// TwinCAT 3 PLC project MainPLC
// Title: IrrigationSystem
// Company: CleanGreens Solutions SA
// ProjectVersion: 0.5beat1
// ProgramVersion: 3.1.4024.0
// libraries:
//   CL_CleanGreensObjectsLibrary, * (CleanGreens SA)
//   CmpBitmapPool, * (System)
//   Tc2_Database, * (Beckhoff Automation GmbH)
//   Tc2_DataExchange, * (Beckhoff Automation GmbH)
//   Tc2_IoFunctions, * (Beckhoff Automation GmbH)
//   Tc2_Math, * (Beckhoff Automation GmbH)
//   Tc2_MC2, * (Beckhoff Automation GmbH)
//   Tc2_Standard, * (Beckhoff Automation GmbH)
//   Tc2_SUPS, * (Beckhoff Automation GmbH)
//   Tc2_System, * (Beckhoff Automation GmbH)
//   Tc2_TcpIp, * (Beckhoff Automation GmbH)
//   Tc2_Utilities, * (Beckhoff Automation GmbH)
//   Tc2_XmlDataSrv, * (Beckhoff Automation GmbH)
//   Tc3_Database, * (Beckhoff Automation GmbH)
//   Tc3_EventLogger, * (Beckhoff Automation GmbH)
//   Tc3_IotBase, * (Beckhoff Automation GmbH)
//   Tc3_IotCommunicator, * (Beckhoff Automation GmbH)
//   Tc3_JsonXml, * (Beckhoff Automation GmbH)
//   Tc3_Module, * (Beckhoff Automation GmbH)
//   VisuDialogs, * (System)
//   VisuSymbols, * (System)
//   VisuUserMgmt, * (System)
//   VisuSymbols,3.5.10.0,System
// project tree:
//   DUTs/ E_AxisErrorType.TcDUT, ST_Analog_HWI.TcDUT (not stored), ST_AXIS_MOVE_PROFILE.TcDUT, ST_CardState_HWI.TcDUT, ST_ChannelAX8206_HWI.TcDUT, ST_DriverAX8206_HWI.TcDUT, ST_PositioningLaser_HWI.TcDUT (not stored), ST_PwrSupplyAX8620_HWI.TcDUT (not stored), ST_RobotLineBoxTest_HWI.TcDUT, ST_Robot_HWI.TcDUT, ST_SystemStatus_ARP.TcDUT, ST_SystemStatus_AR.TcDUT, E_RequAxle.TcDUT, E_StepMC.TcDUT, ST_AxisMC.TcDUT, ST_Robot_Axes.TcDUT, ST_SystemStatus.TcDUT (not stored), ST_SystemStatus_ARR.TcDUT
//   GVLs/ C.TcGVL, CBot.TcGVL, G.TcGVL, GVL.TcGVL
//   / PlcTask.TcTTO
//   POUs/AxisDay2Training/ CL_Axis_old.TcPOU, FB_AxisStMachine.TcPOU, FB_AxisStMachineMaster.TcPOU
//   POUs/ CL_AxisDriverAX8206.TcPOU, CL_AxisDriverL1LeftBack.TcPOU, CL_AxisDriverL1LeftFront.TcPOU, CL_AxisDriverL2RightFront.TcPOU, CL_AxisDriverL2RightBack.TcPOU, CL_AxisMC.TcPOU, CL_AxisMCMaster.TcPOU, CL_AxisMCL2RightBack.TcPOU, CL_AxisMCL1LeftFront.TcPOU, CL_AxisMCL1LeftBack.TcPOU, CL_AxisMCL2RightFront.TcPOU, CL_CardCom.TcPOU, CL_CGSSystemBase.TcPOU, FB_testAxleAllJog.TcPOU, FB_PowerAxis1.TcPOU, FB_PowerMaster.TcPOU, FB_testAxisL1LeftFrontJog.TcPOU, FB_testAxleMasterJog.TcPOU, Main.TcPOU
// real-time tasks:
//   TASK PlcTask: cycle T#10ms, priority 20, ADS port 350
//   TASK VISU_TASK: cycle T#200000us, priority 30, ADS port 351
// motion (NC):
//   TASK NC-Task 1 SAF: cycle T#2ms, priority 4, ADS port 501
//   TASK NC-Task 1 SVB: cycle T#10ms, priority 8, ADS port 511
//   AXIS CGSMini_R01AxisL1LeftBack (id 6)
//     General: UnitName=m
//     Dynamic: AccelerationMaximum=0.5, DecelerationMaximum=1.5, Acceleration=0.3, Deceleration=1, Jerk=0.33
//     Velo: RefSearch=0.01752, RefSync=0.01752, SlowManual=0.0876, FastManual=0.5256, Fast=1.752, Maximum=0.67
//     OtherSettings: AllowMotionCmdToSlave=true
//     encoder EncType=19
//       EncPara: ScaleFactorNumerator=0.79, ScaleFactorDenominator=26214400, Inverse=true, MaxCount=#xffffffff
//         ActPosCorrection: Enable=true, Time=1
//     drive DrvType=16
//       DrvPara: Inverse=true, MaxCount=#xffffffff, DriveControlDWord=#x00020100
//         Analog: VeloReferenz=0.737, VeloScale=71.5255737304688, TorqueSetpointScale=10, ScaleFactorActTorque=0.1
//         TimeComp: TaskDelayCycles=1
//     controller CtrType=1
//       CtrPara: PriorControlFactor=1
//         PosDiffControl: Range=0.1
//         Observer: BandWidth=20
//   AXIS CGSMini_R01AxisL2RightFront (id 7)
//     General: UnitName=m
//     Dynamic: AccelerationMaximum=0.5, DecelerationMaximum=1.5, Acceleration=0.3, Deceleration=1, Jerk=0.33
//     Velo: RefSearch=0.01752, RefSync=0.01752, SlowManual=0.0876, FastManual=0.5256, Fast=1.752, Maximum=0.67
//     OtherSettings: AllowMotionCmdToSlave=true
//     encoder EncType=19
//       EncPara: ScaleFactorNumerator=0.79, ScaleFactorDenominator=26214400, Inverse=true, MaxCount=#xffffffff
//         ActPosCorrection: Enable=true, Time=1
//     drive DrvType=16
//       DrvPara: Inverse=true, MaxCount=#xffffffff, DriveControlDWord=#x00020100
//         Analog: VeloReferenz=0.737, VeloScale=71.5255737304688, TorqueSetpointScale=10, ScaleFactorActTorque=0.1
//         TimeComp: TaskDelayCycles=1
//     controller CtrType=1
//       CtrPara: PriorControlFactor=1
//         PosDiffControl: Range=0.1
//         Observer: BandWidth=20
//   AXIS CGSMini_R01AxisL2RightBack (id 8)
//     General: UnitName=m
//     Dynamic: AccelerationMaximum=0.5, DecelerationMaximum=1.5, Acceleration=0.3, Deceleration=1, Jerk=0.33
//     Velo: RefSearch=0.01752, RefSync=0.01752, SlowManual=0.0876, FastManual=0.5256, Fast=1.752, Maximum=0.67
//     OtherSettings: AllowMotionCmdToSlave=true
//     encoder EncType=19
//       EncPara: ScaleFactorNumerator=0.79, ScaleFactorDenominator=26214400, Inverse=true, MaxCount=#xffffffff
//         ActPosCorrection: Enable=true, Time=1
//     drive DrvType=16
//       DrvPara: Inverse=true, MaxCount=#xffffffff, DriveControlDWord=#x00020100
//         Analog: VeloReferenz=0.737, VeloScale=71.5255737304688, TorqueSetpointScale=10, ScaleFactorActTorque=0.1
//         TimeComp: TaskDelayCycles=1
//     controller CtrType=1
//       CtrPara: PriorControlFactor=1
//         PosDiffControl: Range=0.1
//         Observer: BandWidth=20
//   AXIS CGSMini_R01AxisL1LeftFront (id 5)
//     General: UnitName=m
//     Dynamic: AccelerationMaximum=0.5, DecelerationMaximum=1.5, Acceleration=0.3, Deceleration=1, Jerk=0.33
//     Velo: RefSearch=0.01752, RefSync=0.01752, SlowManual=0.0876, FastManual=0.5256, Fast=1.752, Maximum=0.67
//     OtherSettings: AllowMotionCmdToSlave=true
//     encoder EncType=19
//       EncPara: ScaleFactorNumerator=0.79, ScaleFactorDenominator=26214400, Inverse=true, MaxCount=#xffffffff
//         ActPosCorrection: Enable=true, Time=1
//     drive DrvType=16
//       DrvPara: Inverse=true, MaxCount=#xffffffff, DriveControlDWord=#x00020100
//         Analog: VeloReferenz=0.737, VeloScale=71.5255737304688, TorqueSetpointScale=10, ScaleFactorActTorque=0.1
//         TimeComp: TaskDelayCycles=1
//     controller CtrType=1
//       CtrPara: PriorControlFactor=1
//         PosDiffControl: Range=0.1
//         Observer: BandWidth=20
//   AXIS CGSMini_R01AxisMaster (id 14)
//     General: UnitName=m
//     Dynamic: AccelerationMaximum=0.5, DecelerationMaximum=1.5, Acceleration=0.3, Deceleration=1, Jerk=0.33
//     Velo: RefSearch=0.01752, RefSync=0.01752, SlowManual=0.0876, FastManual=0.5256, Fast=1.752, Maximum=0.67
//     OtherSettings: AllowMotionCmdToSlave=true
//     encoder EncType=1
//       EncPara: ScaleFactorNumerator=0.79, ScaleFactorDenominator=26214400, Inverse=true
//         ActPosCorrection: Enable=true, Time=1
//     drive DrvType=5
//       DrvPara: Inverse=true
//         Analog: VeloReferenz=0.737, TorqueSetpointScale=10, ScaleFactorActTorque=0.1
//         TimeComp: TaskDelayCycles=1
//     controller CtrType=1
//       CtrPara: PriorControlFactor=1
//         PosDiffControl: Range=0.1
//         Observer: BandWidth=20
//   AXIS Sim_Robot01AxisLine1Back (id 9)
//     OtherSettings: AllowMotionCmdToSlave=true
//     encoder EncType=1
//     drive DrvType=5
//       Analog: TorqueSetpointScale=10, ScaleFactorActTorque=0.1
//       TimeComp: TaskDelayCycles=1
//     controller CtrType=1
//       CtrPara: PriorControlFactor=1
//         Observer: BandWidth=20
//   AXIS Sim_Robot01AxisLine2Back (id 10)
//     OtherSettings: AllowMotionCmdToSlave=true
//     encoder EncType=1
//     drive DrvType=5
//       Analog: TorqueSetpointScale=10, ScaleFactorActTorque=0.1
//       TimeComp: TaskDelayCycles=1
//     controller CtrType=1
//       CtrPara: PriorControlFactor=1
//         Observer: BandWidth=20
//   AXIS Sim_Robot01AxisLine1Front (id 11)
//     OtherSettings: AllowMotionCmdToSlave=true
//     encoder EncType=1
//     drive DrvType=5
//       Analog: TorqueSetpointScale=10, ScaleFactorActTorque=0.1
//       TimeComp: TaskDelayCycles=1
//     controller CtrType=1
//       CtrPara: PriorControlFactor=1
//         Observer: BandWidth=20
//   AXIS Sim_Robot01AxisLine2Front (id 12)
//     OtherSettings: AllowMotionCmdToSlave=true
//     encoder EncType=1
//     drive DrvType=5
//       Analog: TorqueSetpointScale=10, ScaleFactorActTorque=0.1
//       TimeComp: TaskDelayCycles=1
//     controller CtrType=1
//       CtrPara: PriorControlFactor=1
//         Observer: BandWidth=20
//   AXIS Sim_Robot01AxisMaster (id 13)
//     OtherSettings: AllowMotionCmdToSlave=true
//     encoder EncType=1
//     drive DrvType=5
//       Analog: TorqueSetpointScale=10, ScaleFactorActTorque=0.1
//       TimeComp: TaskDelayCycles=1
//     controller CtrType=1
//       CtrPara: PriorControlFactor=1
//         Observer: BandWidth=20
// I/O:
//   DEVICE CGSMini_IRSMainPLCSafe, AmsNetId 5.93.147.0.2.1
//     CGSMini_RobotAllMainCab-EL1200 [EK1200-5000 EtherCAT Power supply (2A E-Bus)]
//       CGSMini_RobotAllLicenses-EL6070 [EL6070 1Ch. Licensing-Terminal]
//       CGSMini_Robot01LineBoxOverCurrProt1-EL9222 [EL9222-5500 Overcurrent protection 24V DC, 2Ch., max. 10A (sum), adjustable]
//       CGSMini_Robot01LineBoxOutN01-EL2008 [EL2008 8Ch. Dig. Output 24V, 0.5A]
//       CGSMini_RobotAllMainCabInN01-EL1008 [EL1008 8Ch. Dig. Input 24V, 3ms]
//       CGSMini_Robot01LineBoxInN01-EL1008 [EL1008 8Ch. Dig. Input 24V, 3ms]
//       CGSMini_Robot01LineBoxAnaInN01-EL3202 [EL3202 2Ch. Ana. Input PT100 (RTD)]
//       CGSMini_Robot01LineBoxAnaInN02-EL3054 [EL3054 4Ch. Ana. Input 4-20mA]
//       CGSMini_Robot01LineBoxAnaInN03-EL3202 [EL3202 2Ch. Ana. Input PT100 (RTD)]
//       CGSMini_Robot01LineBoxSafeInN01-EL1918 [EL1918, 8Ch. Safety Input 24V, TwinSAFE] (disabled)
//         modules: Module 1 (FSOE), Module 2 (FSLOGIC)
//       CGSMini_Robot01LineBoxInN02-EL1004tmp [EL1004 4Ch. Dig. Input 24V, 3ms]
//       CGSMini_Robot01LineBoxInN03-EL1004tmp [EL1004 4Ch. Dig. Input 24V, 3ms]
//       CGSMini_RobotAllMainCabAnaInN01-EL3443 [EL3443 3Ch. Power Measuring]
//       CGSMini_Robot01MainCabEtherCATBusEK1122 [EK1122 2 port EtherCAT junction]
//         CGSMini_Robot01Laser-SickDL100 [DL100]
//         CGSMini_Robot01OnboardBox-EK1100 [EK1100 EtherCAT Coupler (2A E-Bus)]
//           CGSMini_Robot01OnBoardBoxOutN01-EL2008 [EL2008 8Ch. Dig. Output 24V, 0.5A]
//           CGSMini_Robot01OnBoardBoxAnaInN04-EL3054 [EL3054 4Ch. Ana. Input 4-20mA]
//           CGSMini_Robot01OnBoardBoxEndBus-EL9011 [EL9011 End Terminal]
//         CGSMini_Robot01OnboardAxisPwrSupply-AX8620 [AX8620-0000-0105]
//           CGSMini_Robot01OnboardAxisDriverL2Right-AX8206 [AX8206-0200-0104 (2Ch. 6A servo axis, safe-motion)]
//             modules: Device, Device, Device, Device, Device, Device, Device, Device, Device, Device, Device (Safety), Device, Device, Device, Device, Device, Device, Device, Device, Device, Device, Device, Device, Device, Device, Device, Device, Device, Device, Device, Device, Back, Back, Back, Back, Back, Back, Back, Back, Back, Back, Back, Back, Back, Back, Back, Back, Back, Back, Back, Back, Back, Back, Back, Back, Back, Back, Back, Front, Front, Front, Front, Front, Front, Front, Front, Front, Front, Front, Front, Front, Front, Front, Front, Front, Front, Front, Front, Front, Front, Front, Front, Front, Front, Front
//             startup 12992:1 := 414D383733312D78437830 // Ch A Motor parameters / Configured motor type
//             startup 24768:0 := FEFF // Ch A Interpolation sub mode select
//             startup 13000:5 := 0200 // Ch A Motor thermal model / Reaction
//             startup 13000:6 := 0000C841 // Ch A Motor thermal model / Partial fraction factor
//             startup 12992:12 := 00803B45 // Ch A Motor parameters / Motor rated speed
//             startup 12992:13 := 8D97A63F // Ch A Motor parameters / Motor rated torque
//             startup 24694:0 := 5A050000 // Ch A Motor standstill torque
//             startup 24800:0 := D007 // Ch A Positive torque/force limit value
//             startup 24801:0 := D007 // Ch A Negative torque/force limit value
//             startup 12288:6 := 4158383230362D303230302D30303030 // Ch A AxisMain parameters / Configured drive type
//             startup 12867:1 := 0000803F // Ch A TorqueCtrl parameters / Configured channel rated current
//             startup 12867:2 := 00004040 // Ch A TorqueCtrl parameters / Configured channel peak current
//             startup 24672:0 := 08 // Ch A Modes of operation
//             startup 12864:1 := 0D4DF043 // Ch A TorqueCtrl parameters mappable / Torque control proportional gain q
//             startup 12864:2 := 8A0E7C39 // Ch A TorqueCtrl parameters mappable / Torque control integral action time q
//             startup 12608:1 := 3C03B63C // Ch A VeloCtrl parameters mappable / Velocity control proportional gain
//             startup 12608:2 := 6F12033C // Ch A VeloCtrl parameters mappable / Velocity control integral action time
//             startup 12608:3 := 00701446 // Ch A VeloCtrl parameters mappable / Bipolar velocity limit value
//             startup 12992:15 := 0100 // Ch A Motor parameters / Motor temperature sensor connection
//             startup 12611:4 := 0400 // Ch A VeloCtrl observer / Observer type
//             startup 24672:0 := 08 // Ch A Modes of operation
//             startup 12296:2 := 00 // Ch A AxisMain parameters encoder polarity / Primary encoder actual values
//             startup 14016:1 := 414D383733312D78437830 // Ch B Motor parameters / Configured motor type
//             startup 26816:0 := FEFF // Ch B Interpolation sub mode select
//             startup 14024:5 := 0200 // Ch B Motor thermal model / Reaction
//             startup 14024:6 := 0000C841 // Ch B Motor thermal model / Partial fraction factor
//             startup 14016:12 := 00803B45 // Ch B Motor parameters / Motor rated speed
//             startup 14016:13 := 8D97A63F // Ch B Motor parameters / Motor rated torque
//             startup 26742:0 := 5A050000 // Ch B Motor standstill torque
//             startup 26848:0 := D007 // Ch B Positive torque/force limit value
//             startup 26849:0 := D007 // Ch B Negative torque/force limit value
//             startup 13312:6 := 4158383230362D303230302D30303030 // Ch B AxisMain parameters / Configured drive type
//             startup 13891:1 := 0000803F // Ch B TorqueCtrl parameters / Configured channel rated current
//             startup 13891:2 := 00004040 // Ch B TorqueCtrl parameters / Configured channel peak current
//             startup 26720:0 := 08 // Ch B Modes of operation
//             startup 13888:1 := 0D4DF043 // Ch B TorqueCtrl parameters mappable / Torque control proportional gain q
//             startup 13888:2 := 8A0E7C39 // Ch B TorqueCtrl parameters mappable / Torque control integral action time q
//             startup 13632:1 := 3C03B63C // Ch B VeloCtrl parameters mappable / Velocity control proportional gain
//             startup 13632:2 := 6F12033C // Ch B VeloCtrl parameters mappable / Velocity control integral action time
//             startup 13632:3 := 00701446 // Ch B VeloCtrl parameters mappable / Bipolar velocity limit value
//             startup 14016:15 := 0100 // Ch B Motor parameters / Motor temperature sensor connection
//             startup 13635:4 := 0400 // Ch B VeloCtrl observer / Observer type
//             startup 26720:0 := 08 // Ch B Modes of operation
//             startup 13320:2 := 00 // Ch B AxisMain parameters encoder polarity / Primary encoder actual values
//           CGSMini_Robot01OnboardAxisDriverL1Left-AX8206 [AX8206-0200-0104 (2Ch. 6A servo axis, safe-motion)]
//             modules: Device, Device, Device, Device, Device, Device, Device, Device, Device, Device, Device (Safety), Device, Device, Device, Device, Device, Device, Device, Device, Device, Device, Device, Device, Device, Device, Device, Device, Device, Device, Device, Device, Back, Back, Back, Back, Back, Back, Back, Back, Back, Back, Back, Back, Back, Back, Back, Back, Back, Back, Back, Back, Back, Back, Back, Back, Back, Back, Back, Front, Front, Front, Front, Front, Front, Front, Front, Front, Front, Front, Front, Front, Front, Front, Front, Front, Front, Front, Front, Front, Front, Front, Front, Front, Front, Front
//             startup 12992:1 := 414D383733312D78437830 // Ch A Motor parameters / Configured motor type
//             startup 24768:0 := FEFF // Ch A Interpolation sub mode select
//             startup 13000:5 := 0200 // Ch A Motor thermal model / Reaction
//             startup 13000:6 := 0000C841 // Ch A Motor thermal model / Partial fraction factor
//             startup 12992:12 := 00803B45 // Ch A Motor parameters / Motor rated speed
//             startup 12992:13 := 8D97A63F // Ch A Motor parameters / Motor rated torque
//             startup 24694:0 := 5A050000 // Ch A Motor standstill torque
//             startup 24800:0 := D007 // Ch A Positive torque/force limit value
//             startup 24801:0 := D007 // Ch A Negative torque/force limit value
//             startup 12288:6 := 4158383230362D303230302D30303030 // Ch A AxisMain parameters / Configured drive type
//             startup 12867:1 := 0000803F // Ch A TorqueCtrl parameters / Configured channel rated current
//             startup 12867:2 := 00004040 // Ch A TorqueCtrl parameters / Configured channel peak current
//             startup 24672:0 := 08 // Ch A Modes of operation
//             startup 12864:1 := 0D4DF043 // Ch A TorqueCtrl parameters mappable / Torque control proportional gain q
//             startup 12864:2 := 8A0E7C39 // Ch A TorqueCtrl parameters mappable / Torque control integral action time q
//             startup 12608:1 := 3C03B63C // Ch A VeloCtrl parameters mappable / Velocity control proportional gain
//             startup 12608:2 := 6F12033C // Ch A VeloCtrl parameters mappable / Velocity control integral action time
//             startup 12608:3 := 00701446 // Ch A VeloCtrl parameters mappable / Bipolar velocity limit value
//             startup 12992:15 := 0100 // Ch A Motor parameters / Motor temperature sensor connection
//             startup 12611:4 := 0400 // Ch A VeloCtrl observer / Observer type
//             startup 24672:0 := 08 // Ch A Modes of operation
//             startup 12296:2 := 00 // Ch A AxisMain parameters encoder polarity / Primary encoder actual values
//             startup 14016:1 := 414D383733312D78437830 // Ch B Motor parameters / Configured motor type
//             startup 26816:0 := FEFF // Ch B Interpolation sub mode select
//             startup 14024:5 := 0200 // Ch B Motor thermal model / Reaction
//             startup 14024:6 := 0000C841 // Ch B Motor thermal model / Partial fraction factor
//             startup 14016:12 := 00803B45 // Ch B Motor parameters / Motor rated speed
//             startup 14016:13 := 8D97A63F // Ch B Motor parameters / Motor rated torque
//             startup 26742:0 := 5A050000 // Ch B Motor standstill torque
//             startup 26848:0 := D007 // Ch B Positive torque/force limit value
//             startup 26849:0 := D007 // Ch B Negative torque/force limit value
//             startup 13312:6 := 4158383230362D303230302D30303030 // Ch B AxisMain parameters / Configured drive type
//             startup 13891:1 := 0000803F // Ch B TorqueCtrl parameters / Configured channel rated current
//             startup 13891:2 := 00004040 // Ch B TorqueCtrl parameters / Configured channel peak current
//             startup 26720:0 := 08 // Ch B Modes of operation
//             startup 13888:1 := 0D4DF043 // Ch B TorqueCtrl parameters mappable / Torque control proportional gain q
//             startup 13888:2 := 8A0E7C39 // Ch B TorqueCtrl parameters mappable / Torque control integral action time q
//             startup 13632:1 := 3C03B63C // Ch B VeloCtrl parameters mappable / Velocity control proportional gain
//             startup 13632:2 := 6F12033C // Ch B VeloCtrl parameters mappable / Velocity control integral action time
//             startup 13632:3 := 00701446 // Ch B VeloCtrl parameters mappable / Bipolar velocity limit value
//             startup 14016:15 := 0100 // Ch B Motor parameters / Motor temperature sensor connection
//             startup 13635:4 := 0400 // Ch B VeloCtrl observer / Observer type
//             startup 26720:0 := 08 // Ch B Modes of operation
//             startup 13320:2 := 00 // Ch B AxisMain parameters encoder polarity / Primary encoder actual values
//           CGSMini_Robot01OnBoardBoxEndBus1-EL9011 [EL9011 End Terminal]
// variable links:
//   MainPLC/MainPLC Instance <-> CGSMini_IRSMainPLCSafe/CGSMini_RobotAllMainCab-EL1200/CGSMini_Robot01LineBoxAnaInN01-EL3202
//     PlcTask Inputs/G.stBoxIN/stAnaInN01_3202State/bNotValid <-> WcState/WcState
//     PlcTask Inputs/G.stBoxIN/stAnaInN01_3202State/uiDataState <-> InfoData/State
//   MainPLC/MainPLC Instance <-> CGSMini_IRSMainPLCSafe/CGSMini_RobotAllMainCab-EL1200/CGSMini_Robot01LineBoxAnaInN02-EL3054
//     PlcTask Inputs/G.stBoxIN/stAnaInN02_3054State/bNotValid <-> WcState/WcState
//     PlcTask Inputs/G.stBoxIN/stAnaInN02_3054State/uiDataState <-> InfoData/State
//   MainPLC/MainPLC Instance <-> CGSMini_IRSMainPLCSafe/CGSMini_RobotAllMainCab-EL1200/CGSMini_Robot01LineBoxAnaInN03-EL3202
//     PlcTask Inputs/G.stBoxIN/stAnaInN03_3202State/bNotValid <-> WcState/WcState
//     PlcTask Inputs/G.stBoxIN/stAnaInN03_3202State/uiDataState <-> InfoData/State
//   MainPLC/MainPLC Instance <-> CGSMini_IRSMainPLCSafe/CGSMini_RobotAllMainCab-EL1200/CGSMini_Robot01LineBoxInN01-EL1008
//     PlcTask Inputs/G.stBoxIN/stInN01_1008State/bNotValid <-> WcState/WcState
//     PlcTask Inputs/G.stBoxIN/stInN01_1008State/uiDataState <-> InfoData/State
//   MainPLC/MainPLC Instance <-> CGSMini_IRSMainPLCSafe/CGSMini_RobotAllMainCab-EL1200/CGSMini_Robot01LineBoxInN02-EL1004tmp
//     PlcTask Inputs/G.stBoxIN/stInN02_1004State/bNotValid <-> WcState/WcState
//     PlcTask Inputs/G.stBoxIN/stInN02_1004State/uiDataState <-> InfoData/State
//   MainPLC/MainPLC Instance <-> CGSMini_IRSMainPLCSafe/CGSMini_RobotAllMainCab-EL1200/CGSMini_Robot01LineBoxInN03-EL1004tmp
//     PlcTask Inputs/G.stBoxIN/stInN03_1004State/bNotValid <-> WcState/WcState
//     PlcTask Inputs/G.stBoxIN/stInN03_1004State/uiDataState <-> InfoData/State
//   MainPLC/MainPLC Instance <-> CGSMini_IRSMainPLCSafe/CGSMini_RobotAllMainCab-EL1200/CGSMini_Robot01LineBoxOutN01-EL2008
//     PlcTask Inputs/G.stBoxIN/stOutN01_2008State/bNotValid <-> WcState/WcState
//     PlcTask Inputs/G.stBoxIN/stOutN01_2008State/uiDataState <-> InfoData/State
//   MainPLC/MainPLC Instance <-> CGSMini_IRSMainPLCSafe/CGSMini_RobotAllMainCab-EL1200/CGSMini_Robot01LineBoxOverCurrProt1-EL9222
//     PlcTask Inputs/G.stBoxIN/stOverCProt1_9222State/bNotValid <-> WcState/WcState
//     PlcTask Inputs/G.stBoxIN/stOverCProt1_9222State/uiDataState <-> InfoData/State
//   MainPLC/MainPLC Instance <-> CGSMini_IRSMainPLCSafe/CGSMini_RobotAllMainCab-EL1200/CGSMini_Robot01LineBoxSafeInN01-EL1918
//     PlcTask Inputs/G.stBoxIN/stSafety_1918State/bNotValid <-> WcState/WcState
//     PlcTask Inputs/G.stBoxIN/stSafety_1918State/uiDataState <-> InfoData/State
//   MainPLC/MainPLC Instance <-> CGSMini_IRSMainPLCSafe/CGSMini_RobotAllMainCab-EL1200/CGSMini_Robot01MainCabEtherCATBusEK1122/CGSMini_Robot01Laser-SickDL100
//     PlcTask Inputs/G.stBoxIN/stLaserPos_State/bNotValid <-> WcState/WcState
//     PlcTask Inputs/G.stBoxIN/stLaserPos_State/uiDataState <-> InfoData/State
//     PlcTask Inputs/G.stIN/stLaserPos <-> Distance/Distance
//     PlcTask Inputs/G.stIN/stLaserPos_State/bNotValid <-> WcState/WcState
//     PlcTask Inputs/G.stIN/stLaserPos_State/uiDataState <-> InfoData/State
//   MainPLC/MainPLC Instance <-> CGSMini_IRSMainPLCSafe/CGSMini_RobotAllMainCab-EL1200/CGSMini_Robot01MainCabEtherCATBusEK1122/CGSMini_Robot01OnboardAxisPwrSupply-AX8620
//     PlcTask Inputs/G.stIN/stPwrSupplyAX8620/comState/bNotValid <-> WcState/WcState
//     PlcTask Inputs/G.stIN/stPwrSupplyAX8620/comState/uiDataState <-> InfoData/State
//     PlcTask Inputs/G.stIN/stPwrSupplyAX8620/sdiDcInputShift <-> InfoData/DcInputShift
//     PlcTask Inputs/G.stIN/stPwrSupplyAX8620/sdiDcOutputShift <-> InfoData/DcOutputShift
//   MainPLC/MainPLC Instance <-> CGSMini_IRSMainPLCSafe/CGSMini_RobotAllMainCab-EL1200/CGSMini_Robot01MainCabEtherCATBusEK1122/CGSMini_Robot01OnboardAxisPwrSupply-AX8620/CGSMini_Robot01OnboardAxisDriverL1Left-AX8206
//     PlcTask Inputs/G.stIN/stDriverL1Left/comState <-> InfoData/State
//     PlcTask Inputs/G.stIN/stDriverL1Left/sdiDcInputShift <-> InfoData/DcInputShift
//     PlcTask Inputs/G.stIN/stDriverL1Left/sdiDcOutputShift <-> InfoData/DcOutputShift
//   MainPLC/MainPLC Instance <-> CGSMini_IRSMainPLCSafe/CGSMini_RobotAllMainCab-EL1200/CGSMini_Robot01MainCabEtherCATBusEK1122/CGSMini_Robot01OnboardAxisPwrSupply-AX8620/CGSMini_Robot01OnboardAxisDriverL2Right-AX8206
//     PlcTask Inputs/G.stIN/stDriverL2Right/comState <-> InfoData/State
//     PlcTask Inputs/G.stIN/stDriverL2Right/sdiDcInputShift <-> InfoData/DcInputShift
//     PlcTask Inputs/G.stIN/stDriverL2Right/sdiDcOutputShift <-> InfoData/DcOutputShift
//   MainPLC/MainPLC Instance <-> CGSMini_IRSMainPLCSafe/CGSMini_RobotAllMainCab-EL1200/CGSMini_Robot01MainCabEtherCATBusEK1122/CGSMini_Robot01OnboardBox-EK1100
//     PlcTask Inputs/G.stIN/stOnboardBox_1100State/uiDataState <-> InfoData/State
//   MainPLC/MainPLC Instance <-> CGSMini_IRSMainPLCSafe/CGSMini_RobotAllMainCab-EL1200/CGSMini_Robot01MainCabEtherCATBusEK1122/CGSMini_Robot01OnboardBox-EK1100/CGSMini_Robot01OnBoardBoxAnaInN04-EL3054
//     PlcTask Inputs/G.stIN/stAnaInN04_3054State/bNotValid <-> WcState/WcState
//     PlcTask Inputs/G.stIN/stAnaInN04_3054State/uiDataState <-> InfoData/State
//     PlcTask Inputs/G.stIN/stAnaOnboardSpare1/bTError <-> Spare1/Status/Error
//     PlcTask Inputs/G.stIN/stAnaOnboardSpare1/bTLimit1 <-> Spare1/Status/Limit 1
//     PlcTask Inputs/G.stIN/stAnaOnboardSpare1/bTLimit2 <-> Spare1/Status/Limit 2
//     PlcTask Inputs/G.stIN/stAnaOnboardSpare1/bTOverRange <-> Spare1/Status/Overrange
//     PlcTask Inputs/G.stIN/stAnaOnboardSpare1/bTUnderRange <-> Spare1/Status/Underrange
//     PlcTask Inputs/G.stIN/stAnaOnboardSpare1/siAnaRaw <-> Spare1/Value
//   MainPLC/MainPLC Instance <-> CGSMini_IRSMainPLCSafe/CGSMini_RobotAllMainCab-EL1200/CGSMini_Robot01MainCabEtherCATBusEK1122/CGSMini_Robot01OnboardBox-EK1100/CGSMini_Robot01OnBoardBoxOutN01-EL2008
//     PlcTask Inputs/G.stIN/stOutN01_2008State/bNotValid <-> WcState/WcState
//     PlcTask Inputs/G.stIN/stOutN01_2008State/uiDataState <-> InfoData/State
//   MainPLC/MainPLC Instance <-> NC-Task 1 SAF/Axes/CGSMini_R01AxisL1LeftBack
//     PlcTask Inputs/G.stAX.L1LeftBack.NcToPlc <-> Outputs/ToPlc
//     PlcTask Outputs/G.stAX.L1LeftBack.PlcToNc <-> Inputs/FromPlc
//   MainPLC/MainPLC Instance <-> NC-Task 1 SAF/Axes/CGSMini_R01AxisL1LeftFront
//     PlcTask Inputs/G.stAX.L1LeftFront.NcToPlc <-> Outputs/ToPlc
//     PlcTask Outputs/G.stAX.L1LeftFront.PlcToNc <-> Inputs/FromPlc
//   MainPLC/MainPLC Instance <-> NC-Task 1 SAF/Axes/CGSMini_R01AxisL2RightBack
//     PlcTask Inputs/G.stAX.L2RightBack.NcToPlc <-> Outputs/ToPlc
//     PlcTask Outputs/G.stAX.L2RightBack.PlcToNc <-> Inputs/FromPlc
//   MainPLC/MainPLC Instance <-> NC-Task 1 SAF/Axes/CGSMini_R01AxisL2RightFront
//     PlcTask Inputs/G.stAX.L2RightFront.NcToPlc <-> Outputs/ToPlc
//     PlcTask Outputs/G.stAX.L2RightFront.PlcToNc <-> Inputs/FromPlc
//   MainPLC/MainPLC Instance <-> NC-Task 1 SAF/Axes/CGSMini_R01AxisMaster
//     PlcTask Inputs/G.stAX.Master.NcToPlc <-> Outputs/ToPlc
//     PlcTask Outputs/G.stAX.Master.PlcToNc <-> Inputs/FromPlc
//   (this object) <-> CGSMini_IRSMainPLCSafe/CGSMini_RobotAllMainCab-EL1200/CGSMini_Robot01MainCabEtherCATBusEK1122/CGSMini_Robot01OnboardAxisPwrSupply-AX8620/CGSMini_Robot01OnboardAxisDriverL1Left-AX8206
//     Drive/Inputs/In/nDataIn1 <-> Back/Ch A PositionControl Inputs/Ch A Following error actual value
//     Drive/Inputs/In/nDcOutputTime <-> InfoData/DcOutputShift
//     Drive/Inputs/In/nState1 <-> Back/Ch A AxisMain Inputs/Ch A Statusword
//     Drive/Inputs/In/nState2 <-> Back/Ch A AxisMain Inputs/Ch A Statusword @bit 8
//     Drive/Outputs/Out/nCtrl1 <-> Back/Ch A AxisMain Outputs/Ch A Controlword
//     Drive/Outputs/Out/nCtrl2 <-> Back/Ch A AxisMain Outputs/Ch A Controlword @bit 8
//     Drive/Outputs/Out/nDataOut1 <-> Back/Ch A Interpolator Outputs/Ch A Target position
//     Drive/Outputs/Out/nDataOut2 <-> Back/Ch A Interpolator Outputs/Ch A Target velocity
//     Enc/Inputs/In/nDataIn1 <-> Back/Ch A AxisMain Inputs/Ch A Position actual value
//     Enc/Inputs/In/nDcInputTime <-> InfoData/DcInputShift
//     Enc/Inputs/In/nState2 @bit 5 <-> Back/Ch A AxisMain Inputs/Position actual value invalid
//     Drive/Inputs/In/nDataIn1 <-> Front/Ch B PositionControl Inputs/Ch B Following error actual value
//     Drive/Inputs/In/nState1 <-> Front/Ch B AxisMain Inputs/Ch B Statusword
//     Drive/Inputs/In/nState2 <-> Front/Ch B AxisMain Inputs/Ch B Statusword @bit 8
//     Drive/Outputs/Out/nCtrl1 <-> Front/Ch B AxisMain Outputs/Ch B Controlword
//     Drive/Outputs/Out/nCtrl2 <-> Front/Ch B AxisMain Outputs/Ch B Controlword @bit 8
//     Drive/Outputs/Out/nDataOut1 <-> Front/Ch B Interpolator Outputs/Ch B Target position
//     Drive/Outputs/Out/nDataOut2 <-> Front/Ch B Interpolator Outputs/Ch B Target velocity
//     Enc/Inputs/In/nDataIn1 <-> Front/Ch B AxisMain Inputs/Ch B Position actual value
//     Enc/Inputs/In/nState2 @bit 5 <-> Front/Ch B AxisMain Inputs/Position actual value invalid
//   (this object) <-> CGSMini_IRSMainPLCSafe/CGSMini_RobotAllMainCab-EL1200/CGSMini_Robot01MainCabEtherCATBusEK1122/CGSMini_Robot01OnboardAxisPwrSupply-AX8620/CGSMini_Robot01OnboardAxisDriverL2Right-AX8206
//     Drive/Inputs/In/nDataIn1 <-> Front/Ch B PositionControl Inputs/Ch B Following error actual value
//     Drive/Inputs/In/nDcOutputTime <-> InfoData/DcOutputShift
//     Drive/Inputs/In/nState1 <-> Front/Ch B AxisMain Inputs/Ch B Statusword
//     Drive/Inputs/In/nState2 <-> Front/Ch B AxisMain Inputs/Ch B Statusword @bit 8
//     Drive/Outputs/Out/nCtrl1 <-> Front/Ch B AxisMain Outputs/Ch B Controlword
//     Drive/Outputs/Out/nCtrl2 <-> Front/Ch B AxisMain Outputs/Ch B Controlword @bit 8
//     Drive/Outputs/Out/nDataOut1 <-> Front/Ch B Interpolator Outputs/Ch B Target position
//     Drive/Outputs/Out/nDataOut2 <-> Front/Ch B Interpolator Outputs/Ch B Target velocity
//     Enc/Inputs/In/nDataIn1 <-> Front/Ch B AxisMain Inputs/Ch B Position actual value
//     Enc/Inputs/In/nDcInputTime <-> InfoData/DcInputShift
//     Enc/Inputs/In/nState2 @bit 5 <-> Front/Ch B AxisMain Inputs/Position actual value invalid
//     Drive/Inputs/In/nDataIn1 <-> Back/Ch A PositionControl Inputs/Ch A Following error actual value
//     Drive/Inputs/In/nState1 <-> Back/Ch A AxisMain Inputs/Ch A Statusword
//     Drive/Inputs/In/nState2 <-> Back/Ch A AxisMain Inputs/Ch A Statusword @bit 8
//     Drive/Outputs/Out/nCtrl1 <-> Back/Ch A AxisMain Outputs/Ch A Controlword
//     Drive/Outputs/Out/nCtrl2 <-> Back/Ch A AxisMain Outputs/Ch A Controlword @bit 8
//     Drive/Outputs/Out/nDataOut1 <-> Back/Ch A Interpolator Outputs/Ch A Target position
//     Drive/Outputs/Out/nDataOut2 <-> Back/Ch A Interpolator Outputs/Ch A Target velocity
//     Enc/Inputs/In/nDataIn1 <-> Back/Ch A AxisMain Inputs/Ch A Position actual value
//     Enc/Inputs/In/nState2 @bit 5 <-> Back/Ch A AxisMain Inputs/Position actual value invalid
//   __THIS__ <-> MainPLC/MainPLC Instance
//     Inputs/FromPlc <-> PlcTask Outputs/G.stAxes.Line1Back.PlcToNc
//     Inputs/FromPlc <-> PlcTask Outputs/G.stAxes.Line2Back.PlcToNc
//     Outputs/ToPlc <-> PlcTask Inputs/G.stAxes.Line1Back.NcToPlc
//     Outputs/ToPlc <-> PlcTask Inputs/G.stAxes.Line2Back.NcToPlc
//     Inputs/FromPlc <-> PlcTask Outputs/GIQ_Robot01.stAxes.Line1Back.PlcToNc
//     Inputs/FromPlc <-> PlcTask Outputs/GIQ_Robot01.stAxes.Line2Back.PlcToNc
//     Outputs/ToPlc <-> PlcTask Inputs/GIQ_Robot01.stAxes.Line1Back.NcToPlc
//     Outputs/ToPlc <-> PlcTask Inputs/GIQ_Robot01.stAxes.Line2Back.NcToPlc
//     Inputs/FromPlc <-> PlcTask Outputs/G.stAxes.Line1Front.PlcToNc
//     Inputs/FromPlc <-> PlcTask Outputs/G.stAxes.Line2Front.PlcToNc
//     Outputs/ToPlc <-> PlcTask Inputs/G.stAxes.Line1Front.NcToPlc
//     Outputs/ToPlc <-> PlcTask Inputs/G.stAxes.Line2Front.NcToPlc
//     Inputs/FromPlc <-> PlcTask Outputs/GIQ_Robot01.stAxes.Line1Front.PlcToNc
//     Inputs/FromPlc <-> PlcTask Outputs/GIQ_Robot01.stAxes.Line2Front.PlcToNc
//     Outputs/ToPlc <-> PlcTask Inputs/GIQ_Robot01.stAxes.Line1Front.NcToPlc
//     Outputs/ToPlc <-> PlcTask Inputs/GIQ_Robot01.stAxes.Line2Front.NcToPlc
//     Inputs/FromPlc <-> PlcTask Outputs/G.stAxes.Master.PlcToNc
//     Outputs/ToPlc <-> PlcTask Inputs/G.stAxes.Master.NcToPlc
//   (this object) <-> MainPLC/MainPLC Instance
//     Inputs/FromPlc <-> PlcTask Outputs/G.stAxes.Line1Back.PlcToNc
//     Inputs/FromPlc <-> PlcTask Outputs/G.stAxes.Line2Back.PlcToNc
//     Outputs/ToPlc <-> PlcTask Inputs/G.stAxes.Line1Back.NcToPlc
//     Outputs/ToPlc <-> PlcTask Inputs/G.stAxes.Line2Back.NcToPlc
//     Inputs/FromPlc <-> PlcTask Outputs/G.stAxes.Line1Front.PlcToNc
//     Inputs/FromPlc <-> PlcTask Outputs/G.stAxes.Line2Front.PlcToNc
//     Outputs/ToPlc <-> PlcTask Inputs/G.stAxes.Line1Front.NcToPlc
//     Outputs/ToPlc <-> PlcTask Inputs/G.stAxes.Line2Front.NcToPlc
//     Inputs/FromPlc <-> PlcTask Outputs/G.stAxes.Master.PlcToNc
//     Outputs/ToPlc <-> PlcTask Inputs/G.stAxes.Master.NcToPlc
//   (this object) <-> CGSMini_IRSMainPLCSafe
//     CGSMini_RobotAllMainCab-EL1200/CGSMini_Robot01MainCabEtherCATBusEK1122/CGSMini_Robot01OnboardAxisPwrSupply-AX8620/CGSMini_Robot01OnboardAxisDriverL1Left-AX8206/Device/DeviceMain Outputs/Power supply controlword <-> CGSMini_RobotAllMainCab-EL1200/CGSMini_Robot01MainCabEtherCATBusEK1122/CGSMini_Robot01OnboardAxisPwrSupply-AX8620/PSM Controlword for axis/Controlword for axis
//     CGSMini_RobotAllMainCab-EL1200/CGSMini_Robot01MainCabEtherCATBusEK1122/CGSMini_Robot01OnboardAxisPwrSupply-AX8620/CGSMini_Robot01OnboardAxisDriverL2Right-AX8206/Device/DeviceMain Outputs/Power supply controlword <-> CGSMini_RobotAllMainCab-EL1200/CGSMini_Robot01MainCabEtherCATBusEK1122/CGSMini_Robot01OnboardAxisPwrSupply-AX8620/PSM Controlword for axis/Controlword for axis
//     CGSMini_RobotAllMainCab-EL1200/CGSMini_Robot01MainCabEtherCATBusEK1122/CGSMini_Robot01OnboardAxisPwrSupply-AX8620/PSM Controlword for axis/Controlword for axis <-> CGSMini_RobotAllMainCab-EL1200/CGSMini_Robot01MainCabEtherCATBusEK1122/CGSMini_Robot01OnboardAxisPwrSupply-AX8620/CGSMini_Robot01OnboardAxisDriverL1Left-AX8206/Device/DeviceMain Outputs/Power supply controlword
//     CGSMini_RobotAllMainCab-EL1200/CGSMini_Robot01MainCabEtherCATBusEK1122/CGSMini_Robot01OnboardAxisPwrSupply-AX8620/PSM Controlword for axis/Controlword for axis <-> CGSMini_RobotAllMainCab-EL1200/CGSMini_Robot01MainCabEtherCATBusEK1122/CGSMini_Robot01OnboardAxisPwrSupply-AX8620/CGSMini_Robot01OnboardAxisDriverL2Right-AX8206/Device/DeviceMain Outputs/Power supply controlword

CONFIGURATION MainPLC
    RESOURCE PLC ON TwinCAT3
        TASK PlcTask(INTERVAL := T#10ms, PRIORITY := 20);
        PROGRAM Main WITH PlcTask : Main;
    END_RESOURCE
END_CONFIGURATION

// ---- DUTs/E_AxisErrorType.TcDUT
{attribute 'qualified_only'}
{attribute 'strict'}
TYPE E_AxisErrorType :
(
  NoError := 0,
  MCError := 1,
  Retry := 2,
  Timeout := 3,
  
  NoOp := 255
);
END_TYPE

// ---- DUTs/ST_AXIS_MOVE_PROFILE.TcDUT
TYPE ST_AXIS_MOVE_PROFILE :
STRUCT
	Velo	: REAL := 0;// Velocity
	Acc		: REAL := 0;// Acceleration
	Dec		: REAL := 0;// Deceleration
	Jerk	: REAL := 0;// Jerk
END_STRUCT
END_TYPE

// ---- DUTs/ST_CardState_HWI.TcDUT
TYPE ST_CardState_HWI :
STRUCT
  uiDataState   : UINT;
  bNotValid     : BOOL;//true if data not valid
END_STRUCT
END_TYPE

// ---- DUTs/ST_ChannelAX8206_HWI.TcDUT
TYPE ST_ChannelAX8206_HWI :
STRUCT
  siIGBTTemp    : INT;
  rMotorTemp    : REAL;
  rMotorTorque  : REAL;
  udMotorDIGIns : UDINT;
END_STRUCT
END_TYPE

// ---- DUTs/ST_DriverAX8206_HWI.TcDUT
TYPE ST_DriverAX8206_HWI :
STRUCT
  comState          : ST_CardState_HWI;
  sdiDcOutputShift  : DINT;
  sdiDcInputShift   : DINT;
  
  stFront           : ST_ChannelAX8206_HWI;//ChB
  stBack            : ST_ChannelAX8206_HWI;//ChA
END_STRUCT
END_TYPE

// ---- DUTs/ST_RobotLineBoxTest_HWI.TcDUT
TYPE ST_RobotLineBoxTest_HWI :
STRUCT
  stInN01_1008State       : ST_CardState_HWI;//CGSMini_Robot01LineBoxInN01-EL1008
  stInN02_1004State       : ST_CardState_HWI;//CGSMini_Robot01LineBoxInN02-EL1004tmp
  stInN03_1004State       : ST_CardState_HWI;//CGSMini_Robot01LineBoxInN03-EL1004tmp
  stOutN01_2008State      : ST_CardState_HWI;//CGSMini_Robot01LineBoxOutN01-EL2008
  stAnaInN01_3202State    : ST_CardState_HWI;//CGSMini_Robot01LineBoxAnaInN01-EL3202
  stAnaInN02_3054State    : ST_CardState_HWI;//CGSMini_Robot01LineBoxAnaInN02-EL3054
  stAnaInN03_3202State    : ST_CardState_HWI;//CGSMini_Robot01LineBoxAnaInN03-EL3202
  stOverCProt1_9222State  : ST_CardState_HWI;//CGSMini_Robot01LineBoxOverCurrProt1-EL9222
  stLineBox_1100State     : ST_CardState_HWI;//CGSMini_Robot01LineBoxBox-EK1100 not yet available useful in case of only one PLC for all robots line
  stSafety_1918State      : ST_CardState_HWI;//CGSMini_Robot01LineBoxSafeInN01-EL1918
  stLaserPos_State        : ST_CardState_HWI;//CGSMini_Robot01Laser-SickDL100
END_STRUCT
END_TYPE

// ---- DUTs/ST_Robot_HWI.TcDUT
TYPE ST_Robot_HWI :
STRUCT
  stAnaInN04_3054State    : ST_CardState_HWI;//CGSMini_Robot01OnBoardBoxAnaInN04-EL3054
  stOnboardBox_1100State  : ST_CardState_HWI;//CGSMini_Robot01OnboardBox-EK1100
  stLaserPos_State        : ST_CardState_HWI;//CGSMini_Robot01Laser-SickDL100
  stOutN01_2008State      : ST_CardState_HWI;//CGSMini_Robot01OnBoardBoxOutN01-EL2008
  
  stLaserPos              : ST_PositioningLaser_HWI;//CGSMini_Robot01Laser-SickDL100
  stAnaOnboardSpare1      : ST_Analog_HWI;//CGSMini_Robot01OnBoardBoxAnaInN04-EL3054
  stPwrSupplyAX8620       : ST_PwrSupplyAX8620_HWI;//CGSMini_Robot01OnboardAxisAlim-AX8620
  stDriverL1Left          : ST_DriverAX8206_HWI;
  stDriverL2Right         : ST_DriverAX8206_HWI;
 END_STRUCT
END_TYPE

// ---- DUTs/ST_SystemStatus_ARP.TcDUT
TYPE
  ST_SystemStatus_ARP : POINTER TO ARRAY [0..C.uiNumIrrLinesForHMI_C] OF ST_SystemStatus;
END_TYPE

// ---- DUTs/ST_SystemStatus_AR.TcDUT
TYPE 
  ST_SystemStatus_AR : ARRAY [0..C.uiNumIrrLinesForHMI_C] OF ST_SystemStatus;
END_TYPE

// ---- DUTs/E_RequAxle.TcDUT
{attribute 'qualified_only'}
{attribute 'strict'}
TYPE E_RequAxle :
(
  NoRequ := 0,
  PowerOn := 1,
  PowerOff := 2,
  Reset := 3,
  Jog := 4,
  GearInDyn := 10,
  GearOut := 11,
  Stop := 20,
  Error := 254,
  Idle := 255
);
END_TYPE

// ---- DUTs/E_StepMC.TcDUT
{attribute 'qualified_only'}
{attribute 'strict'}
TYPE E_StepMC :
(
  Init := 1,
  Timeout := 2,
  Busy := 3,
  Done := 4,
  CmdAborted := 5,
  
	//STEPS ABSOLUTE
 	MoveAbs		    := 11,
	EndMoveAbs    := 12,
  
  //STEPS PowerOn
  //PowerOnInit   := 20,
  PowerOnCheckStatusError := 21,
  PowerOnCheckStatus := 22,
  PowerOnRetryError := 23,
  
  //Jog
  //JogInitEnd := 30,
  //JogBusyEnd := 31,
  
	//STEPS STOP
 	Stopping		  := 51,
  //EndStopping   := 52,
	  
	//STEPS HOMING
  InitHoming    := 60,
	Homing			  := 61,
  EndHoming     := 62,
  InitAbortHoming := 63,
  AbortHoming   := 64,
  InitRetryHoming := 65,
  RetryHoming     := 66,
	   
  End := 254,
  NoStep := 255
);
END_TYPE

// ---- DUTs/ST_AxisMC.TcDUT
//Add Library Tc2_MC2
TYPE ST_AxisMC:
STRUCT
	fbPower						        : MC_Power;//Axis function - Power
	fbReset						        : MC_Reset;//Axis function - Reset
	fbSetPosition					    : MC_SetPosition;//Axis function - Set Position
	fbStop							      : MC_Stop;//stop
	//fbHalt							      : MC_Halt;//Halt
	fbMoveJog							    : MC_Jog;//Jog
	fbGearInDyn					      : MC_GearInDyn;//Axis coupling - GearInDyn
	fbGearOut						      : MC_GearOut;//Axis coupling - GearOut
  fbReadStatus              : MC_ReadStatus;
  
	fbReadAxisError				    : MC_ReadAxisError;//Read Axis Error
	fbReadActualPosition			: MC_ReadActualPosition;//Read Actual Position
	fbReadActualVelocity			: MC_ReadActualVelocity;//Read Actual Velocity
  
	fbHome							      : MC_Home;//Home
	fbMoveAbsolute1				    : MC_MoveAbsolute;//	MC_MoveAbsolute1
  fbMoveAbsoluteWheelCheck  : MC_MoveAbsolute;// Add CustomAutomation 07.03.2023: Check du diamètre des roues 
  fbMoveAbsoluteCorrection  : MC_MoveAbsolute;// Add CustomAutomation 07.03.2023: Correction fin de parcours
 	fbMoveRelative					  : MC_MoveRelative;//Move Relative
	fbMoveVelocity					  : MC_MoveVelocity;//Move Velocity
	fbPosCorrectionLimiter    : MC_PositionCorrectionLimiter;//Special extensions - Position Correction Limiter

  //fbReadAxisComponents     : MC_ReadAxisComponents;
  //fbRearReadBoolParameter  : MC_ReadBoolParameter;
END_STRUCT
END_TYPE

// ---- DUTs/ST_Robot_Axes.TcDUT
TYPE ST_Robot_Axes :
STRUCT
  L1LeftFront    : AXIS_REF;//Axis4-Line1-Left Front (ChB) - second Drive in I/O Tree
  L1LeftBack     : AXIS_REF;//Axis3-Line1-Left Back (ChA) - second Drive in I/O Tree
  L2RightFront   : AXIS_REF;//Axis2-Line2-Right Front (ChB) - first Drive in I/O Tree
  L2RightBack    : AXIS_REF;//Axis1-Line2-Right Back (ChA)- first Drive in I/O Tree
  Master         : AXIS_REF;
END_STRUCT
END_TYPE

(*
Old Robot HW Drivers assign table
ChA -> Front
ChB -> Back
Axe1-LA-Left Front-GVL_Intern.arAxe[1] - Drive 8 (AX8206-0200-0104) # 'Ch A'
Axe2-LB-Left Back-GVL_Intern.arAxe[2] - Drive 8 (AX8206-0200-0104) # 'Ch B'
Axe3-RA-Right Front-GVL_Intern.arAxe[3] - Drive 9 (AX8206-0200-0104) # 'Ch A'
Axe4-RB-Right Back-GVL_Intern.arAxe[4] - Drive 9 (AX8206-0200-0104) # 'Ch B'
*)

// ---- DUTs/ST_SystemStatus_ARR.TcDUT
TYPE
  ST_SystemStatus_ARR : REFERENCE TO ARRAY [0..C.uiNumIrrLinesForHMI_C] OF ST_SystemStatus;
END_TYPE

// ---- GVLs/C.TcGVL
{attribute 'qualified_only'}
VAR_GLOBAL CONSTANT 
  uiNumIrrLinesForHMI_C         : UINT := 1;//how many robots are handled by a single PLC/HMI
  uiNumIrrLinesInGreenhouse_C   : UINT := 2;//2 Telegram BOT, one for each line or bay or span of the greenhouse, selected based on line number
END_VAR

// ---- GVLs/CBot.TcGVL
{attribute 'qualified_only'}
VAR_GLOBAL CONSTANT
  tTimeOutAxisMC_C              : TIME := T#3S;
  tTimeOutRobotStop_C           : TIME := T#5S;
  tTimeOutAxisMasterMC_C        : TIME := T#3S;
  uiRetryPowerOnCnt_C           : UINT := 6;
  
  lrAroundZero_C                : LREAL := 0.18; // m/s //used to check if velocity is around 0 m/s
END_VAR

// ---- GVLs/G.TcGVL
{attribute 'qualified_only'}
VAR_GLOBAL
  _stSystemStatus_AR      : ST_SystemStatus_AR;
  stSystemStatus_ARR      : REFERENCE TO ST_SystemStatus_AR := _stSystemStatus_AR;
  
  
  {attribute 'TcNcAxis' := '.L1LeftFront                     := CGSMini_R01AxisL1LeftFront;
                          .L1LeftBack                        := CGSMini_R01AxisL1LeftBack;
                          .L2RightFront                      := CGSMini_R01AxisL2RightFront;
                          .L2RightBack                       := CGSMini_R01AxisL2RightBack;
                          .Master                            := CGSMini_R01AxisMaster'}
  stAX : ST_Robot_Axes;
  
  (*
  {attribute 'TcNcAxis' := '.L1LeftFront                     := Sim_Robot01AxisLine1Front;
                          .L1LeftBack                        := Sim_Robot01AxisLine1Back;
                          .L2RightFront                       := Sim_Robot01AxisLine2Front;
                          .L2RightBack                        := Sim_Robot01AxisLine2Back;
                          .Master                           := Sim_Robot01AxisMaster'}
  stAxes : ST_Robot_Axes;*)
 
  
//{attribute 'TcLinkTo':='TIIB[CGSMini_Robot01Laser-SickDL100]^WcState^WcState'}
//bLaserWcState AT %I*:BOOL;

{attribute 'TcLinkTo':='.stInN01_1008State.uiDataState      := TIIB[CGSMini_Robot01LineBoxInN01-EL1008]^InfoData^State;
                        .stInN01_1008State.bNotValid         := TIIB[CGSMini_Robot01LineBoxInN01-EL1008]^WcState^WcState; 
 
                        .stInN02_1004State.uiDataState      := TIIB[CGSMini_Robot01LineBoxInN02-EL1004tmp]^InfoData^State;
                        .stInN02_1004State.bNotValid         := TIIB[CGSMini_Robot01LineBoxInN02-EL1004tmp]^WcState^WcState; 
                        
                        .stInN03_1004State.uiDataState      := TIIB[CGSMini_Robot01LineBoxInN03-EL1004tmp]^InfoData^State;
                        .stInN03_1004State.bNotValid         := TIIB[CGSMini_Robot01LineBoxInN03-EL1004tmp]^WcState^WcState; 
                        
                        .stOutN01_2008State.uiDataState     := TIIB[CGSMini_Robot01LineBoxOutN01-EL2008]^InfoData^State;
                        .stOutN01_2008State.bNotValid        := TIIB[CGSMini_Robot01LineBoxOutN01-EL2008]^WcState^WcState;
                        .stAnaInN01_3202State.uiDataState   := TIIB[CGSMini_Robot01LineBoxAnaInN01-EL3202]^InfoData^State;
                        .stAnaInN01_3202State.bNotValid      := TIIB[CGSMini_Robot01LineBoxAnaInN01-EL3202]^WcState^WcState; 
                        .stAnaInN02_3054State.uiDataState   := TIIB[CGSMini_Robot01LineBoxAnaInN02-EL3054]^InfoData^State;
                        .stAnaInN02_3054State.bNotValid      := TIIB[CGSMini_Robot01LineBoxAnaInN02-EL3054]^WcState^WcState; 
                        .stAnaInN03_3202State.uiDataState   := TIIB[CGSMini_Robot01LineBoxAnaInN03-EL3202]^InfoData^State;
                        .stAnaInN03_3202State.bNotValid      := TIIB[CGSMini_Robot01LineBoxAnaInN03-EL3202]^WcState^WcState; 
                        .stOverCProt1_9222State.uiDataState := TIIB[CGSMini_Robot01LineBoxOverCurrProt1-EL9222]^InfoData^State;
                        .stOverCProt1_9222State.bNotValid    := TIIB[CGSMini_Robot01LineBoxOverCurrProt1-EL9222]^WcState^WcState;                     
 
                        .stSafety_1918State.uiDataState     := TIIB[CGSMini_Robot01LineBoxSafeInN01-EL1918]^InfoData^State;
                        .stSafety_1918State.bNotValid        := TIIB[CGSMini_Robot01LineBoxSafeInN01-EL1918]^WcState^WcState;

                        .stLaserPos_State.uiDataState       := TIIB[CGSMini_Robot01Laser-SickDL100]^InfoData^State;
                        .stLaserPos_State.bNotValid          := TIIB[CGSMini_Robot01Laser-SickDL100]^WcState^WcState;
                        .stLaserPos.udiDistanceRaw          := TIIB[CGSMini_Robot01Laser-SickDL100]^Distance^Distance'}
stBoxIN AT %I*:ST_RobotLineBoxTest_HWI;
  
{attribute 'TcLinkTo':='.stAnaInN04_3054State.uiDataState   := TIIB[CGSMini_Robot01OnBoardBoxAnaInN04-EL3054]^InfoData^State;
                        .stAnaInN04_3054State.bNotValid      := TIIB[CGSMini_Robot01OnBoardBoxAnaInN04-EL3054]^WcState^WcState;
                        .stOnboardBox_1100State.uiDataState := TIIB[CGSMini_Robot01OnboardBox-EK1100]^InfoData^State;
                        .stOutN01_2008State.uiDataState     := TIIB[CGSMini_Robot01OnBoardBoxOutN01-EL2008]^InfoData^State;
                        .stOutN01_2008State.bNotValid        := TIIB[CGSMini_Robot01OnBoardBoxOutN01-EL2008]^WcState^WcState;
                        
                        .stLaserPos_State.uiDataState       := TIIB[CGSMini_Robot01Laser-SickDL100]^InfoData^State;
                        .stLaserPos_State.bNotValid          := TIIB[CGSMini_Robot01Laser-SickDL100]^WcState^WcState;
                        .stLaserPos.udiDistanceRaw          := TIIB[CGSMini_Robot01Laser-SickDL100]^Distance^Distance;
                        
                        .stAnaOnboardSpare1.bTUnderRange    := TIIB[CGSMini_Robot01OnBoardBoxAnaInN04-EL3054]^Spare1^Status^Underrange;
                        .stAnaOnboardSpare1.bTOverRange     := TIIB[CGSMini_Robot01OnBoardBoxAnaInN04-EL3054]^Spare1^Status^Overrange;
                        .stAnaOnboardSpare1.bTLimit1        := TIIB[CGSMini_Robot01OnBoardBoxAnaInN04-EL3054]^Spare1^Status^Limit 1;
                        .stAnaOnboardSpare1.bTLimit2        := TIIB[CGSMini_Robot01OnBoardBoxAnaInN04-EL3054]^Spare1^Status^Limit 2;
                        .stAnaOnboardSpare1.bTError         := TIIB[CGSMini_Robot01OnBoardBoxAnaInN04-EL3054]^Spare1^Status^Error;
                        .stAnaOnboardSpare1.siAnaRaw        := TIIB[CGSMini_Robot01OnBoardBoxAnaInN04-EL3054]^Spare1^Value;
  
                        .stPwrSupplyAX8620.comState.uiDataState:= TIIB[CGSMini_Robot01OnboardAxisPwrSupply-AX8620]^InfoData^State;
                        .stPwrSupplyAX8620.comState.bNotValid   := TIIB[CGSMini_Robot01OnboardAxisPwrSupply-AX8620]^WcState^WcState;
                        .stPwrSupplyAX8620.sdiDcOutputShift := TIIB[CGSMini_Robot01OnboardAxisPwrSupply-AX8620]^InfoData^DcOutputShift;
                        .stPwrSupplyAX8620.sdiDcInputShift  := TIIB[CGSMini_Robot01OnboardAxisPwrSupply-AX8620]^InfoData^DcInputShift;
                        .stPwrSupplyAX8620.bOverTemp        := TIIB[CGSMini_Robot01OnboardAxisPwrSupply-AX8620]^PSM Warning register^Warning^A2 Device overtemperature;  
                        .stPwrSupplyAX8620.bFanMalfunc      := TIIB[CGSMini_Robot01OnboardAxisPwrSupply-AX8620]^PSM Warning register^Warning^A4 Fan malfunction;
                        .stPwrSupplyAX8620.bUnderVoltage    := TIIB[CGSMini_Robot01OnboardAxisPwrSupply-AX8620]^PSM Warning register^Warning^A6 Mains undervoltage;
                        .stPwrSupplyAX8620.bOverVoltage     := TIIB[CGSMini_Robot01OnboardAxisPwrSupply-AX8620]^PSM Warning register^Warning^A5 Mains overvoltage;
                        
                        .stDriverL1Left.comState             := TIIB[CGSMini_Robot01OnboardAxisPwrSupply-AX8620]^CGSMini_Robot01OnboardAxisDriverL1Left-AX8206^InfoData^State;
                        .stDriverL1Left.sdiDcOutputShift     := TIIB[CGSMini_Robot01OnboardAxisPwrSupply-AX8620]^CGSMini_Robot01OnboardAxisDriverL1Left-AX8206^InfoData^DcOutputShift;
                        .stDriverL1Left.sdiDcInputShift      := TIIB[CGSMini_Robot01OnboardAxisPwrSupply-AX8620]^CGSMini_Robot01OnboardAxisDriverL1Left-AX8206^InfoData^DcInputShift;           
            
                        .stDriverL1Left.stFront.siIGBTTemp      := TIIB[CGSMini_Robot01OnboardAxisPwrSupply-AX8620]^CGSMini_Robot01OnboardAxisDriverL1Left-AX8206^Front^Ch B AxisMain Inputs^IGBT temperature;
                        .stDriverL1Left.stFront.udMotorDIGIns   := TIIB[CGSMini_Robot01OnboardAxisPwrSupply-AX8620]^CGSMini_Robot01OnboardAxisDriverL1Left-AX8206^Front^Ch B AxisMain Inputs^Ch B Digital inputs;   
                        .stDriverL1Left.stFront.rMotorTemp      := TIIB[CGSMini_Robot01OnboardAxisPwrSupply-AX8620]^CGSMini_Robot01OnboardAxisDriverL1Left-AX8206^Front^Ch B SyncServoMotor Inputs^Actual motor temperature;
                        .stDriverL1Left.stFront.rMotorTorque    := TIIB[CGSMini_Robot01OnboardAxisPwrSupply-AX8620]^CGSMini_Robot01OnboardAxisDriverL1Left-AX8206^Front^Ch B TorqueControl Inputs^Ch B Torque/force actual value;
                   
                        .stDriverL1Left.stBack.siIGBTTemp       := TIIB[CGSMini_Robot01OnboardAxisPwrSupply-AX8620]^CGSMini_Robot01OnboardAxisDriverL1Left-AX8206^Back^Ch A AxisMain Inputs^IGBT temperature;                                                
                        .stDriverL1Left.stBack.udMotorDIGIns    := TIIB[CGSMini_Robot01OnboardAxisPwrSupply-AX8620]^CGSMini_Robot01OnboardAxisDriverL1Left-AX8206^Back^Ch A AxisMain Inputs^Ch A Digital inputs;
                        .stDriverL1Left.stBack.rMotorTemp       := TIIB[CGSMini_Robot01OnboardAxisPwrSupply-AX8620]^CGSMini_Robot01OnboardAxisDriverL1Left-AX8206^Back^Ch A SyncServoMotor Inputs^Actual motor temperature; 
                        .stDriverL1Left.stBack.rMotorTorque     := TIIB[CGSMini_Robot01OnboardAxisPwrSupply-AX8620]^CGSMini_Robot01OnboardAxisDriverL1Left-AX8206^Back^Ch A TorqueControl Inputs^Ch A Torque/force actual value;

                        .stDriverL2Right.comState             := TIIB[CGSMini_Robot01OnboardAxisPwrSupply-AX8620]^CGSMini_Robot01OnboardAxisDriverL2Right-AX8206^InfoData^State;
                        .stDriverL2Right.sdiDcOutputShift     := TIIB[CGSMini_Robot01OnboardAxisPwrSupply-AX8620]^CGSMini_Robot01OnboardAxisDriverL2Right-AX8206^InfoData^DcOutputShift;
                        .stDriverL2Right.sdiDcInputShift      := TIIB[CGSMini_Robot01OnboardAxisPwrSupply-AX8620]^CGSMini_Robot01OnboardAxisDriverL2Right-AX8206^InfoData^DcInputShift;      
                 
                        .stDriverL2Right.stFront.siIGBTTemp      := TIIB[CGSMini_Robot01OnboardAxisPwrSupply-AX8620]^CGSMini_Robot01OnboardAxisDriverL2Right-AX8206^Front^Ch B AxisMain Inputs^IGBT temperature;
                        .stDriverL2Right.stFront.udMotorDIGIns   := TIIB[CGSMini_Robot01OnboardAxisPwrSupply-AX8620]^CGSMini_Robot01OnboardAxisDriverL2Right-AX8206^Front^Ch B AxisMain Inputs^Ch B Digital inputs;  
                        .stDriverL2Right.stFront.rMotorTemp      := TIIB[CGSMini_Robot01OnboardAxisPwrSupply-AX8620]^CGSMini_Robot01OnboardAxisDriverL2Right-AX8206^Front^Ch B SyncServoMotor Inputs^Actual motor temperature;
                        .stDriverL2Right.stFront.rMotorTorque    := TIIB[CGSMini_Robot01OnboardAxisPwrSupply-AX8620]^CGSMini_Robot01OnboardAxisDriverL2Right-AX8206^Front^Ch B TorqueControl Inputs^Ch B Torque/force actual value;
                    
                        .stDriverL2Right.stBack.siIGBTTemp       := TIIB[CGSMini_Robot01OnboardAxisPwrSupply-AX8620]^CGSMini_Robot01OnboardAxisDriverL2Right-AX8206^Back^Ch A AxisMain Inputs^IGBT temperature;
                        .stDriverL2Right.stBack.udMotorDIGIns    := TIIB[CGSMini_Robot01OnboardAxisPwrSupply-AX8620]^CGSMini_Robot01OnboardAxisDriverL2Right-AX8206^Back^Ch A AxisMain Inputs^Ch A Digital inputs;                        
                        .stDriverL2Right.stBack.rMotorTemp       := TIIB[CGSMini_Robot01OnboardAxisPwrSupply-AX8620]^CGSMini_Robot01OnboardAxisDriverL2Right-AX8206^Back^Ch A SyncServoMotor Inputs^Actual motor temperature;                       
                        .stDriverL2Right.stBack.rMotorTorque     := TIIB[CGSMini_Robot01OnboardAxisPwrSupply-AX8620]^CGSMini_Robot01OnboardAxisDriverL2Right-AX8206^Back^Ch A TorqueControl Inputs^Ch A Torque/force actual value;'}
  stIN AT %I*:ST_Robot_HWI;
 
  AxisL1LeftFront   : CL_AxisMCL1LeftFront;
  AxisL2RightFront  : CL_AxisMCL2RightFront;
  AxisL1LeftBack    : CL_AxisMCL1LeftBack;
  AxisL2RightBack   : CL_AxisMCL2RightBack;
  AxisMaster        : CL_AxisMCMaster;
END_VAR

// ---- GVLs/GVL.TcGVL
{attribute 'qualified_only'}
//Axis day 2 training
VAR_GLOBAL
	Axis_servoA : AXIS_REF;
	Axis_servoB : AXIS_REF;
	Axis_servoVirtual : AXIS_REF;
	Axis_servo : AXIS_REF; 
END_VAR

// ---- POUs/Main.TcPOU
PROGRAM Main
VAR
 	//fbPowerMaster : FB_PowerMaster;
  //fbPowerAxis1 : FB_PowerAxis1;
  //fbAxisStMachine : FB_AxisStMachine;
  
  //fbAxisJog : FB_testAxisL1LeftFrontJog;
  
  //fbAxisAllJog : FB_testAxleAllJog;
  
  fbAxleMasterJog : FB_testAxleMasterJog;
END_VAR

//Axis day 2 training
//myAxisA(AxisInOut := GVL.Axis_servoA);
//myAxisB(AxisInOut := GVL.Axis_servoB);
//myAxisVirtual(AxisInOut := GVL.Axis_servoVirtual);
//myAxisStepper(AxisInOut := GVL.Axis_servo);
//fbAxisStMachine(AxisInOut := GVL.Axis_servoA);

//fbPowerAxis1();
//fbPowerMaster();

//fbTestAxle();
//fbAxisJog();
//fbAxisAllJog();
fbAxleMasterJog();

END_PROGRAM

// ---- POUs/FB_testAxleMasterJog.TcPOU
FUNCTION_BLOCK FB_testAxleMasterJog  EXTENDS CL_MasterRootClass
VAR
 	stm	: UINT := 10;
  stIRL : ST_LineReference;
  bFW, bBW, b, bContinue, bContinue2 : BOOL := FALSE;
END_VAR

G.AxisL1LeftFront(); 
G.AxisL2RightFront();
G.AxisL1LeftBack();
G.AxisL2RightBack();
G.AxisMaster();

Case01Hysto(stm);
CASE stm OF   
  10:
    stIRL.nThis := 0;
    stIRL.nFixedID := 1;    
    b := G.AxisL1LeftFront.Init(stIrrLine := stIRL, stAxisMotor_P := ADR(G.stAX.L1LeftFront), stAxisMaster_P := ADR(G.stAX.Master), stDriver := ADR(G.stIN.stDriverL1Left));
    b := b AND G.AxisL1LeftBack.Init(stIrrLine := stIRL, stAxisMotor_P := ADR(G.stAX.L1LeftBack), stAxisMaster_P := ADR(G.stAX.Master), stDriver := ADR(G.stIN.stDriverL1Left));
    b := b AND G.AxisL2RightFront.Init(stIrrLine := stIRL, stAxisMotor_P := ADR(G.stAX.L2RightFront), stAxisMaster_P := ADR(G.stAX.Master), stDriver := ADR(G.stIN.stDriverL2Right));
    b := b AND G.AxisL2RightBack.Init(stIrrLine := stIRL, stAxisMotor_P := ADR(G.stAX.L2RightBack), stAxisMaster_P := ADR(G.stAX.Master), stDriver := ADR(G.stIN.stDriverL2Right));
    b := b AND G.AxisMaster.Init(stIrrLine := stIRL, stAxisMaster_P := ADR(G.stAX.Master));
    if b then
      stm := 900;
		END_IF   
  
900:
    IF NOT G.AxisL1LeftFront.IsBusy AND NOT G.AxisL2RightFront.IsBusy AND NOT G.AxisL1LeftBack.IsBusy AND NOT G.AxisL2RightBack.IsBusy THEN
      G.AxisL1LeftFront.RequGearOut();
      G.AxisL2RightFront.RequGearOut();
      G.AxisL1LeftBack.RequGearOut();
      G.AxisL2RightBack.RequGearOut();
      stm := 910;
    END_IF    
  910:
    IF G.AxisL1LeftFront.IsDone AND G.AxisL2RightFront.IsDone AND G.AxisL1LeftBack.IsDone AND G.AxisL2RightBack.IsDone THEN
      stm := 920;
    END_IF   
  920:
    IF NOT G.AxisL1LeftFront.IsError AND NOT G.AxisL2RightFront.IsError AND NOT G.AxisL1LeftBack.IsError AND NOT G.AxisL2RightBack.IsError THEN
      stm := 1000;
    ELSE
      stm := 0;
    END_IF
  
  //ATTENTION: to power-on axis, they MUST be decoupled 
  1000:
    IF NOT G.AxisL1LeftFront.IsBusy AND NOT G.AxisL2RightFront.IsBusy AND NOT G.AxisL1LeftBack.IsBusy AND NOT G.AxisL2RightBack.IsBusy THEN
      G.AxisL1LeftFront.RequPowerOn();
      G.AxisL2RightFront.RequPowerOn();
      G.AxisL1LeftBack.RequPowerOn();
      G.AxisL2RightBack.RequPowerOn();
      stm := 1120;
    END_IF
    
  1120:
    IF G.AxisL1LeftFront.IsDone AND G.AxisL2RightFront.IsDone AND G.AxisL1LeftBack.IsDone AND G.AxisL2RightBack.IsDone THEN
      stm := 1130;
    END_IF
    
  1130:
    IF NOT G.AxisL1LeftFront.IsError AND NOT G.AxisL2RightFront.IsError AND NOT G.AxisL1LeftBack.IsError AND NOT G.AxisL2RightBack.IsError THEN
      stm := 1135;
    ELSE
      stm := 0;
    END_IF
  
  1135:
    if NOT G.AxisMaster.IsBusy then
      G.AxisMaster.RequPowerOn();
      stm := 1140;
		END_IF
    
  1140:
    IF G.AxisMaster.IsDone THEN 
      stm := 1150;
    END_IF
    
  1150:
    IF NOT G.AxisMaster.IsError THEN
      stm := 1160;
    ELSE
      stm := 0;
    END_IF
  
  1160:
    IF NOT G.AxisL1LeftFront.IsBusy AND NOT G.AxisL2RightFront.IsBusy AND NOT G.AxisL1LeftBack.IsBusy AND NOT G.AxisL2RightBack.IsBusy THEN
      G.AxisL1LeftFront.RequGearInDyn();
      G.AxisL2RightFront.RequGearInDyn();
      G.AxisL1LeftBack.RequGearInDyn();
      G.AxisL2RightBack.RequGearInDyn();
      stm := 1170;
    END_IF
  
  1170:
    IF G.AxisL1LeftFront.IsDone AND G.AxisL2RightFront.IsDone AND G.AxisL1LeftBack.IsDone AND G.AxisL2RightBack.IsDone THEN
      stm := 1180;
    end_if
    
  1180:
    IF NOT G.AxisL1LeftFront.IsError AND NOT G.AxisL2RightFront.IsError AND NOT G.AxisL1LeftBack.IsError AND NOT G.AxisL2RightBack.IsError THEN
      stm := 1190;
    ELSE
      stm := 0;
    END_IF 
  
  1190:
    if NOT G.AxisMaster.IsBusy then
      G.AxisMaster.RequJogAxisMaster();
      stm := 1200;
    end_if
   
  1200:
    if G.AxisMaster.IsDone then
      stm := 1210;
    end_if
      
  1210:
    if not G.AxisMaster.IsError then
      stm := 1300;
    end_if

  1300:
    bFW := true;
    bBW := FALSE;
    G.AxisMaster.JogExec(bExecJogFWIn := bFW, bExecJogBWIn := bBW);
    IF NOT bContinue THEN
      stm := 1300;
    else
      stm := 1310;
    end_if
  
  1310:
    G.AxisMaster.JogExec(bExecJogFWIn := false, bExecJogBWIn := false);
    stm := 1311;
    
  1311:
    IF G.AxisL1LeftFront.IsVelocityZero AND G.AxisL2RightFront.IsVelocityZero AND G.AxisL1LeftBack.IsVelocityZero AND  G.AxisL2RightBack.IsVelocityZero THEN
      stm := 1312;//physically stopped
    END_IF
 
  1312:
    bFW := FALSE;
    bBW := TRUE;
    G.AxisMaster.JogExec(bExecJogFWIn := bFW, bExecJogBWIn := bBW);
    IF NOT bContinue2 THEN
      stm := 1312;
    else
      stm := 1320;
    end_if

  1320:
    IF NOT G.AxisL1LeftFront.IsBusy AND NOT G.AxisL2RightFront.IsBusy AND NOT G.AxisL1LeftBack.IsBusy AND NOT G.AxisL2RightBack.IsBusy and NOT G.AxisMaster.IsBusy THEN
      G.AxisMaster.RequStop();
      G.AxisL1LeftFront.RequStop();
      G.AxisL2RightFront.RequStop();
      G.AxisL1LeftBack.RequStop();
      G.AxisL2RightBack.RequStop();
      stm := 1330;
    END_IF
    
  1330:
    IF G.AxisL1LeftFront.IsDone AND G.AxisL2RightFront.IsDone AND G.AxisL1LeftBack.IsDone AND G.AxisL2RightBack.IsDone THEN
      stm := 1340;
    end_if

  1340:
    IF NOT G.AxisL1LeftFront.IsError AND NOT G.AxisL2RightFront.IsError AND NOT G.AxisL1LeftBack.IsError AND NOT G.AxisL2RightBack.IsError and not G.AxisMaster.IsError THEN
      stm := 1350;
    ELSE
      stm := 0;
    END_IF 

  1350:
    IF G.AxisL1LeftFront.IsStandStill AND G.AxisL2RightFront.IsStandStill AND G.AxisL1LeftBack.IsStandStill AND  G.AxisL2RightBack.IsStandStill AND G.AxisMaster.IsStandStill THEN
      stm := 1400;//physically stopped
    END_IF
  
  1400:
    IF NOT G.AxisL1LeftFront.IsBusy AND NOT G.AxisL2RightFront.IsBusy AND NOT G.AxisL1LeftBack.IsBusy AND NOT G.AxisL2RightBack.IsBusy THEN
      G.AxisL1LeftFront.RequGearOut();
      G.AxisL2RightFront.RequGearOut();
      G.AxisL1LeftBack.RequGearOut();
      G.AxisL2RightBack.RequGearOut();
      stm := 1410;
    END_IF
    
  1410:
    IF G.AxisL1LeftFront.IsDone AND G.AxisL2RightFront.IsDone AND G.AxisL1LeftBack.IsDone AND G.AxisL2RightBack.IsDone THEN
      stm := 1420;
    end_if
    
  1420:
    IF NOT G.AxisL1LeftFront.IsError AND NOT G.AxisL2RightFront.IsError AND NOT G.AxisL1LeftBack.IsError AND NOT G.AxisL2RightBack.IsError THEN
      stm := 0;
    ELSE
      stm := 0;
    END_IF 

  0:; //park 
END_CASE

END_FUNCTION_BLOCK

// ---- POUs/CL_AxisMCL1LeftFront.TcPOU
FUNCTION_BLOCK CL_AxisMCL1LeftFront EXTENDS CL_AxisMC
VAR
  objAxisDriver : CL_AxisDriverL1LeftFront;
END_VAR

SUPER^();

METHOD PUBLIC Init : BOOL
VAR_INPUT
  stIrrLine       : ST_LineReference;
  stAxisMotor_P	  : POINTER TO AXIS_REF;
  stAxisMaster_P  : POINTER TO AXIS_REF;
  stDriver        : POINTER TO ST_DriverAX8206_HWI;
END_VAR
Init := FALSE;
IF stDriver <> 0 THEN
  Init := objAxisDriver.Init(stDriver := stDriver);
  Init := Init AND SUPER^.InitMC(stIrrLine := stIrrLine, stAxisMotor_P := stAxisMotor_P, stAxisMaster_P := stAxisMaster_P, AxisDriver_P := ADR(objAxisDriver));
END_IF
END_METHOD

METHOD PROTECTED InitDefect : BOOL
InitDefect := SUPER^.InitDefect();
ADSLOGSTR(ADSLOG_MSGTYPE_LOG, 'CL_AxisMCL1LeftFront init defect','');
END_METHOD

METHOD PROTECTED InitParams : BOOL
VAR_INPUT
END_VAR
InitParams := SUPER^.InitParams();
_sWhichAxis := 'left(L1)-front';
_lrInverse := 1.0;
END_METHOD

END_FUNCTION_BLOCK

// ---- POUs/CL_AxisMC.TcPOU
FUNCTION_BLOCK CL_AxisMC EXTENDS CL_CGSSystemBase
VAR
  bInit                 : BOOL := FALSE;
  _AxisDriver_R         : REFERENCE TO CL_AxisDriverAX8206;
  _stMotorAxis_R			  : REFERENCE TO AXIS_REF;//axis reference linked to I/O
  _stMasterAxis_R       : REFERENCE TO AXIS_REF;//master axis
  _stMC                 : ST_AxisMC;
  
  _stAxisJog_R          : REFERENCE TO AXIS_REF;
  
  //private properties 
  _nStep                : E_StepMC;
  _nStepMain            : E_RequAxle := E_RequAxle.Idle;
  
  _nRequAxle            : E_RequAxle;
  _nPreviousRequ        : E_RequAxle;
  _nActualRequ          : E_RequAxle;  
  
  _bIsDone			        : BOOL := FALSE;	
  _bIsBusy			        : BOOL := FALSE;	
  _bIsPowered			      : BOOL := FALSE;
	_bError			          : BOOL := FALSE;
  _bIsAxisMaster			  : BOOL := FALSE;
	_nErrorId		          : UDINT := 0;
 
  //remove the following after debug
  _bMCBusy			        : BOOL;
  _bMCError			        : BOOL;
  _bMCStatus            : BOOL;
	//_MCerrId			        : UDINT;

  _bPowerOn             : BOOL := FALSE;
  _bGearOut             : BOOL := FALSE;
  _bStop                : BOOL := FALSE;
  _bGearInDyn           : BOOL := FALSE;
  _bJogFW               : BOOL := FALSE;
  _bJogBW               : BOOL := FALSE;
  _bIsCoupled           : BOOL := FALSE;
  _bEnableEntryMC       : BOOL := FALSE;
  
  _bReadStatusOK        : BOOL := FALSE;
  _bReadVelOK           : BOOL := FALSE;
  _bReadPosOK           : BOOL := FALSE;
  
  _bExecPreviousRequ    : BOOL := FALSE;
    
	//_bEnableMove          : BOOL := TRUE;   // Enable the moving of axis
	_lrAxisOverride	      : LREAL:= 100.0;  // Override of the axis velocity
  
  _lrActPos             : LREAL;
  _lrActVel             : LREAL;
  
  //_bExecJog             : BOOL := FALSE;
  //_bExecJogFWIn         : BOOL := FALSE;
  // _bExecJogBWIn         : BOOL := FALSE;
  _bJogCmdAborted       : BOOL := FALSE;
  _bAxisMovedbyJog      : BOOL := FALSE;

  _lrJogVelocity        : LREAL;
  
  _bGearInCmdAborted    : BOOL := FALSE;
  _lrMotorGearRatio     : LREAL;
  _lrAcceleration       : LREAL;
  _lrInverse            : LREAL; //Line1-Left -> _lrInverse:=1.0 while Line2-Right -> _lrInverse:=-1.0
  
  stStopProfile         : ST_AXIS_MOVE_PROFILE; //.Dec If the value is 0, the deceleration from the move command is used   .Jerk If the value is 0, the deceleration from the move command is used
 
  //counters
  _uiRetryPowerOnCnt_C  : UINT := CBot.uiRetryPowerOnCnt_C;  //PowerOn retry
  _uiRetryPowerOnCnt    : UINT := _uiRetryPowerOnCnt_C;  //_uiRetryPowerOnCnt_C PowerOn retry
   
  //timeout MC request
  _bRequTimeout         : BOOL;
  WaitNextState         : CL_WaitTimer; 
  
  _nJogMode             : E_JogMode;
  
  //Error handling
  //_bErrMsgShow        : BOOL := true;
  _sWhichAxis           : STRING(16);
  _nAxisErrType         : E_AxisErrorType;
END_VAR

IF bInit THEN
  THIS^.RunEntryMC();
  THIS^.RunMC();//run M.otion C.ontrol (MC) FB function on entry
  THIS^.Run();
  THIS^.RunMC();//run M.otion C.ontrol (MC) FB function on exit, to speed-up 1 PLC cycle the refresh of the MC command
END_IF

METHOD PROTECTED InitDefect : BOOL
VAR_INPUT
END_VAR
InitDefect := true;
END_METHOD

METHOD PUBLIC InitMC : BOOL
VAR_INPUT
  stIrrLine       : ST_LineReference;
  stAxisMotor_P	  : POINTER TO AXIS_REF;
  stAxisMaster_P  : POINTER TO AXIS_REF;
  AxisDriver_P    : POINTER TO CL_AxisDriverAX8206;
END_VAR
InitMC := FALSE;
//do not check AxisDriver_P, because master axis ha no driver associated
IF stAxisMotor_P <> 0 AND stAxisMaster_P <> 0 AND NOT bInit THEN
  _bIsAxisMaster := stAxisMotor_P = stAxisMaster_P;
  
  _stMotorAxis_R REF= stAxisMotor_P^;
  _stMasterAxis_R REF= stAxisMaster_P^;
  _stAxisJog_R REF= _stMotorAxis_R;
  
  IF _bIsAxisMaster THEN
    bInit := AxisDriver_P = 0; 
    //do not assign _AxisDriver_R, because master axis has no driver associated !
  ELSE
    bInit := TRUE;
    _AxisDriver_R REF= AxisDriver_P^;
	END_IF
  
  bInit := binit AND SUPER^.InitSystemBase( IrrLine := stIrrLine, stSystemStatus_ARR := G.stSystemStatus_ARR);
  bInit := bInit AND InitParams();
  bInit := bInit AND InitDefect();
  InitMC := bInit;
  
  _bEnableEntryMC := TRUE;//read entry MC continuosly
END_IF
END_METHOD

METHOD PROTECTED InitParams : BOOL
VAR_INPUT
END_VAR
InitParams := true;
//if the listed parameters are equal 0.0 -> the standard parameter from the axis configuration in the System Manager is used
_lrJogVelocity := 0.3;//m/s
_nJogMode := MC_JOGMODE_STANDARD_SLOW;//MC_JOGMODE_STANDARD_FAST;  MC_JOGMODE_CONTINUOUS
_nJogMode := MC_JOGMODE_STANDARD_FAST; 
_stMC.fbMoveJog(Axis := _stMotorAxis_R, Position := 0.0, Velocity := _lrJogVelocity, Acceleration := 0.0, Deceleration := 0.0, Jerk := 0.0);
_lrInverse := 1.0;
END_METHOD

PROPERTY IsBusy : bool
GET
IsBusy := _bIsBusy;
END_GET
END_PROPERTY

PROPERTY PUBLIC IsCoupled : BOOL
GET
IsCoupled := _stMotorAxis_R.Status.Coupled and not _bIsAxisMaster;//_bIsAxisMaster1 must be never coupled!
END_GET
END_PROPERTY

PROPERTY IsDone : bool
GET
IsDone := _bIsDone;
END_GET
END_PROPERTY

PROPERTY IsDoneNoError : bool
GET
IsDoneNoError := _bIsDone and not _bError;
END_GET
END_PROPERTY

PROPERTY PUBLIC IsError : Bool
GET
IsError := _bError;
END_GET
END_PROPERTY

PROPERTY PUBLIC IsStandStill : BOOL
GET
IsStandStill := _stMotorAxis_R.Status.StandStill;
END_GET
END_PROPERTY

PROPERTY PUBLIC IsVelocityZero : BOOL
GET
IsVelocityZero := _lrActVel < CBot.lrAroundZero_C and _lrActVel > -CBot.lrAroundZero_C;
END_GET
END_PROPERTY

METHOD PUBLIC JogExec : BOOL
VAR_INPUT
  //bExecIn : BOOL := FALSE;
  bExecJogFWIn : BOOL := FALSE;
  bExecJogBWIn : BOOL := FALSE;
END_VAR
if bExecJogFWIn <> bExecJogBWIn then
  _bJogFW := bExecJogFWIn;
  _bJogBW := bExecJogBWIn;
else
  _bJogFW := _bJogBW := FALSE;
END_IF
 _bAxisMovedbyJog := _stMC.fbMoveJog.Active;
 _bJogCmdAborted := _stMC.fbMoveJog.CommandAborted;
END_METHOD

PROPERTY PUBLIC nErrorID : UDINT
GET
nErrorID := _nErrorID;
END_GET
END_PROPERTY

METHOD PRIVATE OnEntryRequ
VAR_INPUT
END_VAR
_nStep := E_StepMC.Init;

_bIsBusy := TRUE;
_bIsDone := false;
_bError := FALSE;
_nErrorId	:= 0;

_bRequTimeout := false;
_bGearInCmdAborted := FALSE;
_bJogCmdAborted := false;
_bJogFW := _bJogBW := false;
_bAxisMovedbyJog := false;
//_bExecJogFWIn := _bExecJogBWIn := false;
//_bExecJog := false;
END_METHOD

METHOD PRIVATE OnExitRequError
VAR_INPUT
  ErrorIDIn     : UDINT;
  nAxisErrIn    : E_AxisErrorType;
END_VAR
_nStepMain := E_RequAxle.Error;
_bIsDone	:= TRUE;
_bIsBusy	:= FALSE;
_bError := true;
_nErrorId := ErrorIDIn;
_bExecPreviousRequ := FALSE;
_bIsPowered := FALSE;
_nAxisErrType := nAxisErrIn;
END_METHOD

METHOD PRIVATE OnExitRequOk
VAR_INPUT
END_VAR
_nStepMain := E_RequAxle.Idle;
_bIsDone	:= TRUE;
_bIsBusy	:= FALSE;
_bError := false;
_nErrorId	:= 0;
//_nRequAxle := E_RequAxle.NoRequ;//not necessary set inside method Run
END_METHOD

METHOD PRIVATE OnExitRequRetry
VAR_INPUT
  ErrorIDIn : UDINT;
  RequRetryIn  : E_RequAxle;
END_VAR
_nStepMain := E_RequAxle.Idle;
_bIsDone	:= FALSE;
_bIsBusy	:= TRUE;
_bError := true;
_nErrorId := ErrorIDIn;
_nRequAxle := RequRetryIn;
_bExecPreviousRequ := TRUE;
_bIsPowered := false;
END_METHOD

{attribute 'TcRpcEnable'}
METHOD RequGearInDyn : bool
RequGearInDyn := bInit AND _bIsPowered AND NOT _bError AND NOT _bIsBusy AND NOT _bIsAxisMaster;
//_stMotorAxis_R <> _stMasterAxis_R GearInDyn only on real axis not master axis
//_stMotorAxis_R = _stMasterAxis_R GearInDyn on virtual axis in this case make no sense
IF RequGearInDyn AND NOT _bIsCoupled THEN
	_nRequAxle := E_RequAxle.GearInDyn;
  //request GearInDyn only if the axis is decoupled
else
  //RequGearInDyn can be only false, _bIsCoupled can be true or false
  _bIsDone := _bIsCoupled OR _bIsAxisMaster;
  //the axis was already coupled; only in this case set _bIsDone to true as the request to couple is "virtually" executed
  //otherwise set it to false
  _nRequAxle := E_RequAxle.NoRequ;
END_IF
END_METHOD

{attribute 'TcRpcEnable'}
METHOD RequGearOut : bool
RequGearOut := bInit AND NOT _bError AND NOT _bIsBusy AND NOT _bIsAxisMaster;
//to not check _bIsPowered because the GearOut cab be executed even if not power-on
//_stMotorAxis_R <> _stMasterAxis_R GearInDyn only on real axis not master axis
//_stMotorAxis_R = _stMasterAxis_R GearInDyn on virtual axis in this case make no sense

IF RequGearOut and _bIsCoupled THEN
	_nRequAxle := E_RequAxle.GearOut;
  //request GearOut only if the axis is coupled
else
  //RequGearOut can be only false, _bIsCoupled can be true or false
  _bIsDone := NOT _bIsCoupled OR _bIsAxisMaster;
  //the axis was already Decoupled; only in this case set _bIsDone to true as the request to decouple is "virtually" executed
  //otherwise set it to false
  _nRequAxle := E_RequAxle.NoRequ;
END_IF
END_METHOD

{attribute 'TcRpcEnable'}
METHOD RequJogAxisMaster : bool
RequJogAxisMaster := bInit AND _bIsPowered AND NOT _bError AND NOT _bIsBusy AND _bIsAxisMaster;
IF RequJogAxisMaster THEN
  _stAxisJog_R := _stMasterAxis_R;//change the pointer to the Jog axis ref in order to use the master axis
	_nRequAxle := E_RequAxle.Jog;
else
  _nRequAxle := E_RequAxle.NoRequ;
END_IF
END_METHOD

{attribute 'TcRpcEnable'}
METHOD RequJogAxisMotor : bool
RequJogAxisMotor := bInit and _bIsPowered AND NOT _bError and not _bIsBusy AND NOT _bIsAxisMaster;
IF RequJogAxisMotor THEN
  _stAxisJog_R := _stMotorAxis_R;//change the pointer to the Jog axis ref in order to use the motor axis
	_nRequAxle := E_RequAxle.Jog;
else
  _nRequAxle := E_RequAxle.NoRequ;
END_IF
END_METHOD

{attribute 'TcRpcEnable'}
METHOD RequPowerOFF : BOOL
RequPowerOFF := bInit and _bIsPowered AND NOT _bError and not _bIsBusy;
IF RequPowerOFF THEN
	_nRequAxle := E_RequAxle.PowerOff;
else
  _nRequAxle := E_RequAxle.NoRequ;
END_IF
END_METHOD

{attribute 'TcRpcEnable'}
METHOD RequPowerON : bool
RequPowerON := bInit and NOT _bIsPowered AND NOT _bError and not _bIsBusy;
IF RequPowerON THEN
	_nRequAxle := E_RequAxle.PowerOn;
else
  _nRequAxle := E_RequAxle.NoRequ;
END_IF
END_METHOD

{attribute 'TcRpcEnable'}
METHOD public RequReset : bool
RequReset := bInit;//no conditions: this request is always executed -> removed bInit and NOT _bError and not _bIsBusy
IF bInit THEN
	_nRequAxle	:= E_RequAxle.Reset;
END_IF
END_METHOD

METHOD PRIVATE RequResetAndPrevious : BOOL
RequResetAndPrevious := bInit;//no conditions: this request is always executed -> removed bInit and NOT _bError and not _bIsBusy
IF bInit THEN
	_nRequAxle	:= E_RequAxle.Reset;
  _bExecPreviousRequ := TRUE;
END_IF
END_METHOD

{attribute 'TcRpcEnable'}
METHOD RequStop : bool
RequStop := bInit and _bIsPowered AND NOT _bError and not _bIsBusy;
IF RequStop THEN
	_nRequAxle := E_RequAxle.Stop;
else
  _nRequAxle := E_RequAxle.NoRequ;
END_IF
END_METHOD

METHOD PRIVATE Run
WaitNextState();
CASE _nStepMain OF
  E_RequAxle.Idle:
    IF _nRequAxle <> E_RequAxle.NoRequ THEN
      IF NOT _bExecPreviousRequ THEN
        _nPreviousRequ := _nRequAxle;
      END_IF
      _nStepMain := _nRequAxle;
      _nActualRequ := _nRequAxle;
      _nRequAxle := E_RequAxle.NoRequ;
      OnEntryRequ();
    end_if
  E_RequAxle.PowerOn :    StmPowerOn_Off(bPowerOnIn := TRUE);
  E_RequAxle.PowerOff :   StmPowerOn_Off(bPowerOnIn := FALSE);
  E_RequAxle.Jog :        StmJog();
  E_RequAxle.GearInDyn :  StmGearInDyn();
  E_RequAxle.GearOut :    StmGearOut();
  E_RequAxle.Reset :      StmReset();
  E_RequAxle.Error :      StmError();
  E_RequAxle.Stop :       StmStop();
  else;     
END_CASE
Case01Hysto(_nStepMain);
END_METHOD

METHOD PRIVATE RunEntryMC
//fbReadStatus run only once before to execute all
_stMC.fbReadStatus(Axis:= _stMotorAxis_R,Enable := _bEnableEntryMC,Valid => _bReadStatusOK); //return TRUE, if the states was determined successfully.
//_stMotorAxis_R.Status (struct type ST_AxisStatus) contains extensive status information about an axis. 
//This data structure must be updated in each PLC cycle by calling MC_ReadStatus or by calling the action 
//_stMotorAxis_R.ReadStatus().
//_stMotorAxis_R.Status.MotionState (struct type  MC_AxisStates) contains motion state in the PLCopen state diagram 
//_stMotorAxis_R.NcToPlc.CoupleState.1 for the moment it doesn't work...waiting for an answer _stMotorAxis_R.Status.Coupled doesn't return true even if the axis is coupled
_stMC.fbReadActualVelocity(Axis:= _stMotorAxis_R,Enable := _bEnableEntryMC,Valid => _bReadVelOK, ActualVelocity => _lrActVel);//return TRUE, if the velocity was determined successfully.
_stMC.fbReadActualPosition(Axis:= _stMotorAxis_R,Enable := _bEnableEntryMC,Valid => _bReadPosOK, Position => _lrActPos);//return TRUE, if the position was determined successfully.

_bIsCoupled := _stMotorAxis_R.Status.Coupled;

IF NOT _bReadStatusOK THEN
  ;//add a defect in case the MC_ReadStatus fails
END_IF
IF NOT _bReadVelOK THEN
  ;//add a defect in case it fails    
END_IF
IF NOT _bReadPosOK THEN
  ;//add a defect in case it fails    
END_IF
END_METHOD

METHOD PRIVATE RunMC
_stMC.fbPower(
    Axis:= _stMotorAxis_R, 
    Enable:= _bPowerOn, 
    Enable_Positive:= _bPowerOn, 
    Enable_Negative:= _bPowerOn, 
    Override:= _lrAxisOverride, 
    Status=>_bMCStatus ,
    Busy=>_bMCBusy , 
    Error=>_bMCError);
        
_stMC.fbReset(
    Axis:= _stMotorAxis_R, 
    Busy=>_bMCBusy , 
    Error=>_bMCError);

_stMC.fbMoveJog(
    Axis := _stAxisJog_R,
    JogForward := _bJogFW,
    JogBackwards := _bJogBW,
    Mode := _nJogMode,
    Velocity := _lrJogVelocity);
      
_stMC.fbGearInDyn(
    Master := _stMasterAxis_R,
    Slave:= _stMotorAxis_R,
    Enable := _bGearInDyn,//continous signal true
    GearRatio := _lrMotorGearRatio,
    Acceleration := _lrAcceleration,
    Busy=>_bMCBusy,
    Error=>_bMCError);
//ATTENTION MC_GearInDyn has Busy = Active = true until is active!

_stMC.fbGearOut(
    Slave:= _stMotorAxis_R,
    Execute := _bGearOut);//rising edge

_stMC.fbStop(
    Axis:= _stMotorAxis_R,
    Execute := _bStop);//rising edge
   
///////////////////////////////////////////////OLD
	(*
	fbReadAxisError				    : MC_ReadAxisError;//Status and parameter - Read Axis Error
  
 	fbSetPosition					    : MC_SetPosition;//Axis function - Set Position
	fbHome							      : MC_Home;//Home
	fbMoveAbsolute1				    : MC_MoveAbsolute;//	MC_MoveAbsolute1
  fbMoveAbsoluteWheelCheck  : MC_MoveAbsolute;// Add CustomAutomation 07.03.2023: Check du diamètre des roues 
  fbMoveAbsoluteCorrection  : MC_MoveAbsolute;// Add CustomAutomation 07.03.2023: Correction fin de parcours
 	fbMoveRelative					  : MC_MoveRelative;//Move Relative
	fbMoveVelocity					  : MC_MoveVelocity;//Move Velocity
	fbPosCorrectionLimiter    : MC_PositionCorrectionLimiter;//Special extensions - Position Correction Limiter

_stMC.fbHome(Axis:=MotorAxle^, bCalibrationCam:=_udCalibrationSensor_P^.19,
		    Options := stHomingOption, Position := lrnOffsetExtractorHoming);    
fbMoveAbso(Axis:= _AxisREF_P^);
fbTimeRetryHomming(IN := nStep = E_StepAxis.AbortHoming);
fbTimeAbortHoming(IN := nStep = E_StepAxis.RetryHoming);
fbTrigErrorMotor(CLK := _AxisREF_P^.NcToPlc.ErrorCode <> 0);
*)
END_METHOD

METHOD PRIVATE StmError
var
  nActLine      : UINT;
  fbFormatStr	  : FB_FormatString;
  sTmp          : T_MaxString;
  sOutMsg       : T_MaxString;
  //bTmp1Err      : BOOL;
  //nErrIdOut     : UDINT;
END_VAR
_nStepMain := E_RequAxle.Idle;
//_stMC.fbPower.Enable := FALSE;
//_stMC.fbPower.Enable_Positive	:= FALSE;
//_stMC.fbPower.Enable_Negative	:= FALSE;
//fbHome.Execute := FALSE;
//fbHomeInv.Execute	:= FALSE;

if MRIrrLine <> MRIrrLineFixedID then 
  nActLine := MRIrrLineFixedID;//the real line if an HMI for each ronot is contained in MRIrrLineFixedID
else
  nActLine := MRIrrLine;
END_IF

sTmp := _sWhichAxis;  
fbFormatStr(
  sFormat	:= 'Irrigation line: %d  Axis motor: %s  MC error ID: %d  Request: ', 
  arg1  := F_UINT(nActLine),
  arg2  := F_STRING(sTmp),
  arg3	:= F_UDINT(_nErrorId),
  //bError => bTmp1Err,  
  //nErrId => nErrIdOut, 
  sOut	=> sOutMsg);

sTmp := '';
case _nActualRequ of
  E_RequAxle.PowerOn : sTmp := 'Power ON';
  E_RequAxle.PowerOff : sTmp := 'Power OFF';
  E_RequAxle.Reset : sTmp := 'Reset';
  E_RequAxle.Jog : sTmp := 'Jog';
  E_RequAxle.GearInDyn : sTmp := 'GearInDyn';
  E_RequAxle.GearOut : sTmp := 'GearOut';
  E_RequAxle.Stop : sTmp := 'Stop';
  else
    sTmp := 'Not listed';
end_case
sOutMsg := concat(sOutMsg,sTmp);

sTmp := '';
CASE _nAxisErrType OF
  E_AxisErrorType.NoError : sTmp :=' failed no error reported';
  E_AxisErrorType.MCError : sTmp :=' failed due to MC error';
  E_AxisErrorType.Retry : sTmp :=' failed after retry';
  E_AxisErrorType.Timeout : sTmp :=' timed out';
  ELSE;
END_CASE
sOutMsg := concat(sOutMsg,sTmp);
  
ADSLOGSTR(ADSLOG_MSGTYPE_LOG, 'CL_Axis error loop  %s',sOutMsg);
//ADSLOGSTR(ADSLOG_MSGTYPE_MSGBOX, 'CL_Axis error loop  %s',sOutMsg);
END_METHOD

METHOD PRIVATE StmGearInDyn
CASE _nStep OF 
  E_StepMC.Init :
    _bGearInDyn	:= TRUE;//until enable = true -> As long as "Enable" is TRUE, the gear factor can be changed cyclically
    _bGearOut := false;
    _lrMotorGearRatio := 1.0 * _lrInverse;
    _lrAcceleration := 0.0;// If the value is 0, the standard acceleration from the axis configuration in the System Manager is used
    WaitNextState.Start(CBot.tTimeOutAxisMC_C);
    _nStep := E_StepMC.Busy;
  
  E_StepMC.Busy :
    IF _stMC.fbGearInDyn.CommandAborted THEN
      _nStep := E_StepMC.CmdAborted;
    END_IF
    IF WaitNextState.End THEN
      _nStep := E_StepMC.Timeout;
    ELSIF _stMC.fbGearInDyn.Busy THEN //Active == Busy
      //ATTENTION MC_GearInDyn has Busy = Active = true until is active!
      _nStep := E_StepMC.End;
    END_IF
    
  E_StepMC.End:
    IF NOT _stMC.fbGearInDyn.Error THEN  
      _bIsCoupled := TRUE;
      OnExitRequOk();
    ELSE
      _bRequTimeout := false;
      OnExitRequError(_stMC.fbGearInDyn.ErrorID, E_AxisErrorType.MCError);
    END_IF
  
  E_StepMC.CmdAborted:
    _bGearInCmdAborted := true;
    OnExitRequOk();
    //OnExitRequError(_stMC.fbGearInDyn.ErrorID);
    
  E_StepMC.Timeout:
    _bRequTimeout := true;
    OnExitRequError(_stMC.fbGearInDyn.ErrorID, E_AxisErrorType.Timeout);   
end_case
END_METHOD

METHOD PRIVATE StmGearOut
CASE _nStep OF 
E_StepMC.Init :
  _bGearInDyn	:= FALSE;//disable immediately GearInDyn
  _bGearOut := TRUE; //executed with a rising edge
  WaitNextState.Start(CBot.tTimeOutAxisMC_C);
  _nStep := E_StepMC.Busy;

E_StepMC.Busy :
  IF WaitNextState.End THEN
    _nStep := E_StepMC.Timeout;
  ELSIF NOT _stMC.fbGearOut.Busy THEN
    WaitNextState.Start(CBot.tTimeOutAxisMC_C);
    _nStep := E_StepMC.Done;
  END_IF

E_StepMC.Done :
  IF WaitNextState.End THEN
     _nStep := E_StepMC.Timeout;
  ELSIF _stMC.fbGearOut.Done THEN
    _nStep := E_StepMC.End;
  END_IF
  
E_StepMC.End:
  IF NOT _stMC.fbGearOut.Error THEN  
    _bGearOut := FALSE;//executed with a rising edge
    _bIsCoupled := false;
    OnExitRequOk();
  ELSE
    _bGearOut := false;//executed with a rising edge
    _bRequTimeout := false;
    OnExitRequError(_stMC.fbGearOut.ErrorID, E_AxisErrorType.MCError);
  END_IF

E_StepMC.Timeout:
    _stMC.fbGearOut.Execute := FALSE;
    _bRequTimeout := false;//executed with a rising edge
    OnExitRequError(_stMC.fbGearOut.ErrorID, E_AxisErrorType.Timeout);  
end_case
END_METHOD

METHOD PRIVATE StmJog
CASE _nStep OF 
  E_StepMC.Init://step by default set by OnEntryRequ method
    _bJogFW := false;//_bExecJogFWIn;
    _bJogBW := false;//_bExecJogBWIn;
    _nStep := E_StepMC.Busy;
   
  E_StepMC.Busy :    
    IF _stMC.fbMoveJog.CommandAborted THEN
      _nStep := E_StepMC.CmdAborted;
    ELSIF NOT _stMC.fbMoveJog.Busy THEN
      _nStep := E_StepMC.End;
    END_IF     
        
  E_StepMC.CmdAborted:
    _bAxisMovedbyJog := false;
    _bJogCmdAborted := true;
    OnExitRequOk();
                          
  E_StepMC.End:
    _bJogFW := FALSE;
    _bJogBW := FALSE;
    _bAxisMovedbyJog := FALSE;
    _bJogCmdAborted := false;
    IF NOT _stMC.fbMoveJog.Error THEN  
      OnExitRequOk();
    ELSE
      OnExitRequError(_stMC.fbMoveJog.ErrorID, E_AxisErrorType.MCError);
    end_if                  
end_case
Case02Hysto(_nStep);
END_METHOD

METHOD PRIVATE StmPowerOn_Off
VAR_INPUT
  bPowerOnIn : BOOL;
END_VAR
VAR
  b : BOOL;
END_VAR
CASE _nStep OF   
  E_StepMC.Init:
    _bPowerOn := bPowerOnIn;
    _nStep := E_StepMC.PowerOnCheckStatusError;
  
  E_StepMC.PowerOnCheckStatusError:
    b := _stMotorAxis_R.Status.Error;
    //b := TRUE;
    IF NOT b THEN //really at the level of NC Status Error flag
     _nStep := E_StepMC.PowerOnCheckStatus;
     IF _bIsAxisMaster THEN 
       WaitNextState.Start(CBot.tTimeOutAxisMasterMC_C);
     ELSE
       WaitNextState.Start(CBot.tTimeOutAxisMC_C);
		 END_IF    
     //_uiRetryPowerOnCnt := _uiRetryPowerOnCnt_C; 
    ELSE
      _nStep := E_StepMC.PowerOnRetryError;
 		END_IF
    
  E_StepMC.PowerOnCheckStatus:
    IF bPowerOnIn THEN
      //powering-on
      b := _stMC.fbPower.Status;
    ELSE
      //powering-off
      b := not _stMC.fbPower.Status;
    END_IF
    {IF defined (MiniRobotSim)}
    b := TRUE;
    {END_IF}
    IF b THEN
      b := _stMC.fbPower.Error;
      IF b THEN 
        _nStep := E_StepMC.PowerOnRetryError;
      ELSE       
        _bIsPowered := bPowerOnIn;
        OnExitRequOk();
        _uiRetryPowerOnCnt := _uiRetryPowerOnCnt_C;
        _bExecPreviousRequ := FALSE;
      END_IF
    ELSE 
      IF WaitNextState.End THEN    
        _nStep := E_StepMC.PowerOnRetryError;
      END_IF
    END_IF

  E_StepMC.PowerOnRetryError:
    //_bPowerOn := FALSE;
    IF _uiRetryPowerOnCnt = 0 THEN
      OnExitRequError(_stMC.fbPower.ErrorID, E_AxisErrorType.Retry);//after _uiRetryPowerOnCnt still impossible to PowerOn
      _uiRetryPowerOnCnt := _uiRetryPowerOnCnt_C;
      _bExecPreviousRequ := FALSE;
     ELSE
      OnExitRequRetry(ErrorIDIn := _stMC.fbPower.ErrorID, RequRetryIn := E_RequAxle.Reset);
      _uiRetryPowerOnCnt := _uiRetryPowerOnCnt - 1;
    END_IF    
END_CASE
Case02Hysto(_nStep);
END_METHOD

METHOD PRIVATE StmReset


CASE _nStep OF 
E_StepMC.Init :
  _stMC.fbReset.Execute	:= TRUE;
  WaitNextState.Start(CBot.tTimeOutAxisMC_C);
  _nStep := E_StepMC.Busy;

E_StepMC.Busy :
  IF WaitNextState.End THEN
    _nStep := E_StepMC.Timeout;
  ELSIF _stMC.fbReset.Busy THEN
    WaitNextState.Start(CBot.tTimeOutAxisMC_C);
    _nStep := E_StepMC.Done;
  END_IF

E_StepMC.Done :
  IF WaitNextState.End THEN
     _nStep := E_StepMC.Timeout;
  ELSIF _stMC.fbReset.Done THEN
    _nStep := E_StepMC.End;
  END_IF
  
E_StepMC.End:
  IF NOT _stMC.fbReset.Error THEN  
    _stMC.fbReset.Execute := FALSE;
    IF _bExecPreviousRequ THEN
      _nRequAxle := _nPreviousRequ;
      _nStepMain := E_RequAxle.Idle;
    ELSE
      OnExitRequOk();
    END_IF
  ELSE
    _stMC.fbReset.Execute := FALSE;
    _bRequTimeout := false;
    OnExitRequError(_stMC.fbReset.ErrorID, E_AxisErrorType.MCError);
  END_IF

E_StepMC.Timeout:
    _stMC.fbReset.Execute := FALSE;
    _bRequTimeout := true;
    OnExitRequError(_stMC.fbReset.ErrorID, E_AxisErrorType.Timeout);  
end_case
Case03Hysto(_nStep);
END_METHOD

METHOD PRIVATE StmStop
CASE _nStep OF 
  E_StepMC.Init:
    _bGearInDyn	:= false;
    _stMC.fbStop.Deceleration	:= stStopProfile.Dec;
    _stMC.fbStop.Jerk	:= stStopProfile.Jerk;
    _bStop := true; //executed with a rising edge
    WaitNextState.Start(CBot.tTimeOutAxisMC_C);
    _nStep := E_StepMC.Busy;
  
  E_StepMC.Busy:
    IF WaitNextState.End THEN
      _nStep := E_StepMC.Timeout;
    ELSIF _stMC.fbStop.Busy THEN
      WaitNextState.Start(CBot.tTimeOutRobotStop_C);//this timing is function of the dynamic of the whole robot!
      _nStep := E_StepMC.Stopping;
    END_IF
  
  E_StepMC.Stopping:
     IF WaitNextState.End THEN
      _nStep := E_StepMC.Timeout;
     ELSIF _stMotorAxis_R.Status.NotMoving THEN
       WaitNextState.Start(CBot.tTimeOutAxisMC_C);
      _nStep := E_StepMC.Done;
		 END_IF
     
  E_StepMC.Done:
    IF WaitNextState.End THEN
       _nStep := E_StepMC.Timeout;
    ELSIF _stMC.fbStop.Done THEN
      _nStep := E_StepMC.End;
    END_IF  
    
  E_StepMC.End:
    IF NOT _stMC.fbStop.Error THEN  
      _bStop := false;//executed with a rising edge
      OnExitRequOk();
    ELSE
      _bStop := false;//executed with a rising edge
      _bRequTimeout := false;
      OnExitRequError(_stMC.fbGearOut.ErrorID, E_AxisErrorType.MCError);
    END_IF
  
  E_StepMC.Timeout:
      _bStop := FALSE;
      _bRequTimeout := false;//executed with a rising edge
      OnExitRequError(_stMC.fbGearOut.ErrorID, E_AxisErrorType.Timeout);  
end_case
END_METHOD

END_FUNCTION_BLOCK

// ---- POUs/CL_CGSSystemBase.TcPOU
FUNCTION_BLOCK CL_CGSSystemBase EXTENDS CL_MasterRootClass
VAR
  //INTERNAL VAR
  _stSystemStatus_ARR   : ST_SystemStatus_ARR;
  bInitSysBase          : BOOL := FALSE;
END_VAR

//State machine history
IF bInitSysBase THEN 
  //Manage Mode machine
  IF _stSystemStatus_ARR[MRIrrLine].nRequestModeMachine <> nModeMachine AND _stSystemStatus_ARR[MRIrrLine].nStateMachine = E_StateMachine.cStopped THEN
    _stSystemStatus_ARR[MRIrrLine].nModeMachine := _stSystemStatus_ARR[MRIrrLine].nRequestModeMachine;
  END_IF  
END_IF

METHOD PUBLIC InitSystemBase : BOOL
VAR_INPUT
  //nIrrLine             : UINT := 0;
  //nIrrLineFixedID      : UINT := 0;
  IrrLine              : ST_LineReference;
  stSystemStatus_ARR   : ST_SystemStatus_ARR;
END_VAR
InitSystemBase := FALSE;
IF __ISVALIDREF(stSystemStatus_ARR) AND NOT bInitSysBase 
   AND IrrLine.nThis >= 0 AND IrrLine.nThis <= C.uiNumIrrLinesForHMI_C
   AND IrrLine.nFixedID >= 0 AND IrrLine.nThis <= C.uiNumIrrLinesInGreenhouse_C THEN
    _stSystemStatus_ARR REF= stSystemStatus_ARR;
    MRLineRef := IrrLine;
    InitSystemBase := bInitSysBase := TRUE;
END_IF
END_METHOD

PROPERTY PUBLIC nModeMachine : E_ModeMachine
GET
IF bInitSysBase THEN 
  nModeMachine := _stSystemStatus_ARR[MRIrrLine].nModeMachine;
ELSE
  nModeMachine := E_ModeMachine.Startup;
END_IF
END_GET
SET
IF bInitSysBase THEN 
  _stSystemStatus_ARR[MRIrrLine].nModeMachine := nModeMachine;
ELSE
  _stSystemStatus_ARR[MRIrrLine].nModeMachine := E_ModeMachine.Startup;
END_IF
END_SET
END_PROPERTY

PROPERTY PUBLIC nReqModeMachine : E_ModeMachine
GET
IF bInitSysBase THEN 
  nReqModeMachine := _stSystemStatus_ARR[MRIrrLine].nRequestModeMachine;
ELSE
  nReqModeMachine := E_ModeMachine.Startup;
END_IF
END_GET
SET
IF bInitSysBase THEN 
  _stSystemStatus_ARR[MRIrrLine].nRequestModeMachine := nReqModeMachine;
ELSE
 _stSystemStatus_ARR[MRIrrLine].nRequestModeMachine := E_ModeMachine.Startup;
END_IF
END_SET
END_PROPERTY

PROPERTY PUBLIC nStateMachine : E_StateMachine
GET
IF bInitSysBase THEN 
  nStateMachine := _stSystemStatus_ARR[MRIrrLine].nStateMachine;
ELSE
  nStateMachine := E_StateMachine.cIdle;
END_IF
END_GET
SET
IF bInitSysBase THEN 
  _stSystemStatus_ARR[MRIrrLine].nStateMachine := nStateMachine;
ELSE
  _stSystemStatus_ARR[MRIrrLine].nStateMachine := E_StateMachine.cIdle;;
END_IF
END_SET
END_PROPERTY

METHOD PUBLIC ReqModeMachine : BOOL
VAR_INPUT
  nModeMachine   : E_ModeMachine;;
END_VAR
IF bInitSysBase THEN 
  _stSystemStatus_ARR[MRIrrLine].nRequestModeMachine := nModeMachine;
END_IF
END_METHOD

END_FUNCTION_BLOCK

// ---- POUs/CL_AxisDriverAX8206.TcPOU
FUNCTION_BLOCK CL_AxisDriverAX8206 EXTENDS CL_CardCom
VAR
  bInit                   : BOOL := FALSE;
  _stDriverCom_P          : POINTER TO ST_DriverAX8206_HWI;
  _stDriverCh_P           : POINTER TO ST_ChannelAX8206_HWI;
END_VAR

IF bInit THEN
  THIS^.Run();
END_IF

METHOD PUBLIC IGBTTemp : real
VAR_INPUT
END_VAR
IGBTTemp := INT_TO_REAL(_stDriverCh_P^.siIGBTTemp);
END_METHOD

METHOD PROTECTED InitDefect : BOOL
VAR_INPUT
END_VAR
InitDefect := true;
END_METHOD

METHOD PUBLIC InitDriver : BOOL
VAR_INPUT
  stDriverCom_P     : POINTER TO ST_DriverAX8206_HWI;
  stDriverCh_P      : POINTER TO ST_ChannelAX8206_HWI;
END_VAR
InitDriver := FALSE;
IF stDriverCom_P <> 0 AND stDriverCh_P <> 0 AND NOT bInit THEN
  _stDriverCom_P := stDriverCom_P;
  _stDriverCh_P := stDriverCh_P;
  bInit := InitDriver := InitCom(stCardStateIn_P := ADR(_stDriverCom_P^.comState)) AND  InitDefect() AND InitDefectCom();
END_IF
END_METHOD

METHOD PUBLIC MotorTemp : real
VAR_INPUT
END_VAR
MotorTemp := _stDriverCh_P^.rMotorTemp;
END_METHOD

METHOD PRIVATE Run
VAR_INPUT
END_VAR
END_METHOD

METHOD PUBLIC Torque : REAL
Torque := _stDriverCh_P^.rMotorTorque;
END_METHOD

END_FUNCTION_BLOCK

// ---- POUs/CL_CardCom.TcPOU
FUNCTION_BLOCK CL_CardCom EXTENDS CL_MasterRootClass
VAR
  //private internal methods
  bComInit       : BOOL := FALSE;
  _stCardState_P : POINTER TO ST_CardState_HWI;
END_VAR

IF bComInit THEN
  THIS^.RunCom();
END_IF

METHOD InitCom : BOOL
VAR_INPUT
  stCardStateIn_P : POINTER TO ST_CardState_HWI;
END_VAR
InitCom := false;
_stCardState_P  := stCardStateIn_P;
IF _stCardState_P <> 0 AND NOT bComInit THEN
  bComInit := InitCom := InitDefectCom();
END_IF
END_METHOD

METHOD PROTECTED InitDefectCom : BOOL
VAR_INPUT
END_VAR
InitDefectCom := true;
END_METHOD

METHOD PRIVATE RunCom
VAR_INPUT
END_VAR
END_METHOD

END_FUNCTION_BLOCK

// ---- POUs/CL_AxisDriverL1LeftFront.TcPOU
FUNCTION_BLOCK CL_AxisDriverL1LeftFront EXTENDS CL_AxisDriverAX8206
VAR
END_VAR

SUPER^();

METHOD PUBLIC Init : BOOL
VAR_INPUT  
  stDriver : POINTER TO ST_DriverAX8206_HWI;
END_VAR
Init := FALSE;
IF stDriver <> 0 THEN
  Init := SUPER^.InitDriver(stDriverCom_P := ADR(stDriver^.comState), stDriverCh_P := ADR(stDriver^.stFront));
END_IF
END_METHOD

METHOD PROTECTED InitDefect : BOOL
VAR_INPUT
END_VAR
InitDefect := SUPER^.InitDefect();
ADSLOGSTR(ADSLOG_MSGTYPE_LOG, 'CL_AxisDriverL1LeftFront init defect','');
END_METHOD

END_FUNCTION_BLOCK

// ---- POUs/CL_AxisMCL2RightFront.TcPOU
FUNCTION_BLOCK CL_AxisMCL2RightFront EXTENDS CL_AxisMC
VAR
  objAxisDriver : CL_AxisDriverL2RightFront;
END_VAR

SUPER^();

METHOD PUBLIC Init : BOOL
VAR_INPUT
  stIrrLine       : ST_LineReference;
  stAxisMotor_P	  : POINTER TO AXIS_REF;
  stAxisMaster_P  : POINTER TO AXIS_REF;
  stDriver        : POINTER TO ST_DriverAX8206_HWI;
END_VAR
Init := FALSE;
IF stDriver <> 0 THEN
  Init := objAxisDriver.Init(stDriver := stDriver);
  Init := Init AND SUPER^.InitMC(stIrrLine := stIrrLine, stAxisMotor_P := stAxisMotor_P, stAxisMaster_P := stAxisMaster_P, AxisDriver_P := ADR(objAxisDriver));
END_IF
END_METHOD

METHOD PROTECTED InitDefect : BOOL
InitDefect := SUPER^.InitDefect();
ADSLOGSTR(ADSLOG_MSGTYPE_LOG, 'CL_AxisMCL2RightFront init defect','');
END_METHOD

METHOD PROTECTED InitParams : BOOL
VAR_INPUT
END_VAR
InitParams := SUPER^.InitParams();
_sWhichAxis := 'right(L2)-front';
_lrInverse := -1.0;
END_METHOD

END_FUNCTION_BLOCK

// ---- POUs/CL_AxisDriverL2RightFront.TcPOU
FUNCTION_BLOCK CL_AxisDriverL2RightFront EXTENDS CL_AxisDriverAX8206
VAR
END_VAR

SUPER^();

METHOD PUBLIC Init : BOOL
VAR_INPUT  
  stDriver : POINTER TO ST_DriverAX8206_HWI;
END_VAR
Init := FALSE;
IF stDriver <> 0 THEN
  Init := SUPER^.InitDriver(stDriverCom_P := ADR(stDriver^.comState), stDriverCh_P := ADR(stDriver^.stFront));
END_IF
END_METHOD

METHOD PROTECTED InitDefect : BOOL
VAR_INPUT
END_VAR
InitDefect := SUPER^.InitDefect();
ADSLOGSTR(ADSLOG_MSGTYPE_LOG, 'CL_AxisDriverL2RightFront init defect','');
END_METHOD

END_FUNCTION_BLOCK

// ---- POUs/CL_AxisMCL1LeftBack.TcPOU
FUNCTION_BLOCK CL_AxisMCL1LeftBack EXTENDS CL_AxisMC
VAR
  objAxisDriver : CL_AxisDriverL1LeftBack;
END_VAR

SUPER^();

METHOD PUBLIC Init : BOOL
VAR_INPUT
  stIrrLine       : ST_LineReference;
  stAxisMotor_P	  : POINTER TO AXIS_REF;
  stAxisMaster_P  : POINTER TO AXIS_REF;
  stDriver        : POINTER TO ST_DriverAX8206_HWI;
END_VAR
Init := FALSE;
IF stDriver <> 0 THEN
  Init := objAxisDriver.Init(stDriver := stDriver);
  Init := Init AND SUPER^.InitMC(stIrrLine := stIrrLine, stAxisMotor_P := stAxisMotor_P, stAxisMaster_P := stAxisMaster_P, AxisDriver_P := ADR(objAxisDriver));
END_IF
END_METHOD

METHOD PROTECTED InitDefect : BOOL
InitDefect := SUPER^.InitDefect();
ADSLOGSTR(ADSLOG_MSGTYPE_LOG, 'CL_AxisMCL1LeftBack init defect','');
END_METHOD

METHOD PROTECTED InitParams : BOOL
VAR_INPUT
END_VAR
InitParams := SUPER^.InitParams();
_sWhichAxis := 'left(L1)-back';
_lrInverse := 1.0;
END_METHOD

END_FUNCTION_BLOCK

// ---- POUs/CL_AxisDriverL1LeftBack.TcPOU
FUNCTION_BLOCK CL_AxisDriverL1LeftBack EXTENDS CL_AxisDriverAX8206
VAR
END_VAR

SUPER^();

METHOD PROTECTED InitDefect : BOOL
VAR_INPUT
END_VAR
InitDefect := true;
END_METHOD

END_FUNCTION_BLOCK

// ---- POUs/CL_AxisMCL2RightBack.TcPOU
FUNCTION_BLOCK CL_AxisMCL2RightBack EXTENDS CL_AxisMC
VAR
  objAxisDriver : CL_AxisDriverL2RightBack;
END_VAR

SUPER^();

METHOD PUBLIC Init : BOOL
VAR_INPUT
  stIrrLine       : ST_LineReference;
  stAxisMotor_P	  : POINTER TO AXIS_REF;
  stAxisMaster_P  : POINTER TO AXIS_REF;
  stDriver        : POINTER TO ST_DriverAX8206_HWI;
END_VAR
Init := FALSE;
IF stDriver <> 0 THEN
  Init := objAxisDriver.Init(stDriver := stDriver);
  Init := Init AND SUPER^.InitMC(stIrrLine := stIrrLine, stAxisMotor_P := stAxisMotor_P, stAxisMaster_P := stAxisMaster_P, AxisDriver_P := ADR(objAxisDriver));
END_IF
END_METHOD

METHOD PROTECTED InitDefect : BOOL
InitDefect := SUPER^.InitDefect();
ADSLOGSTR(ADSLOG_MSGTYPE_LOG, 'CL_AxisMCL2RightBack init defect','');
END_METHOD

METHOD PROTECTED InitParams : BOOL
VAR_INPUT
END_VAR
InitParams := SUPER^.InitParams();
_sWhichAxis := 'right(L2)-back';
_lrInverse := -1.0;
END_METHOD

END_FUNCTION_BLOCK

// ---- POUs/CL_AxisDriverL2RightBack.TcPOU
FUNCTION_BLOCK CL_AxisDriverL2RightBack EXTENDS CL_AxisDriverAX8206
VAR
END_VAR

SUPER^();

METHOD PUBLIC Init : BOOL
VAR_INPUT  
  stDriver : POINTER TO ST_DriverAX8206_HWI;
END_VAR
Init := FALSE;
IF stDriver <> 0 THEN
  Init := SUPER^.InitDriver(stDriverCom_P := ADR(stDriver^.comState), stDriverCh_P := ADR(stDriver^.stBack));
END_IF
END_METHOD

METHOD PROTECTED InitDefect : BOOL
VAR_INPUT
END_VAR
InitDefect := SUPER^.InitDefect();
ADSLOGSTR(ADSLOG_MSGTYPE_LOG, 'CL_AxisDriverL2RightBack init defect','');
END_METHOD

END_FUNCTION_BLOCK

// ---- POUs/CL_AxisMCMaster.TcPOU
FUNCTION_BLOCK CL_AxisMCMaster EXTENDS CL_AxisMC
VAR
  //objAxisDriver : CL_AxisDriverMaster; //Axis Master has no hardware driver
END_VAR

SUPER^();

METHOD PUBLIC Init : BOOL
VAR_INPUT
  stIrrLine       : ST_LineReference;
  stAxisMaster_P  : POINTER TO AXIS_REF;
END_VAR
Init := SUPER^.InitMC(stIrrLine := stIrrLine, stAxisMotor_P := stAxisMaster_P, stAxisMaster_P := stAxisMaster_P, AxisDriver_P := 0);
END_METHOD

METHOD PROTECTED InitDefect : BOOL
InitDefect := SUPER^.InitDefect();
ADSLOGSTR(ADSLOG_MSGTYPE_LOG, 'CL_AxisMCMaster init defect','');
END_METHOD

METHOD PROTECTED InitParams : BOOL
VAR_INPUT
END_VAR
InitParams := SUPER^.InitParams();
_sWhichAxis := 'virtual-master';
END_METHOD

END_FUNCTION_BLOCK

// ---- POUs/AxisDay2Training/CL_Axis_old.TcPOU
FUNCTION_BLOCK CL_Axis_old EXTENDS CL_MasterRootClass
VAR_INPUT
	bEnableMove     : BOOL := TRUE;   // Enable the moving of axis
	lrAxisOverride	: LREAL:= 100;    // Override of the axis
END_VAR
VAR_OUTPUT	
	bError			: BOOL := FALSE;
	nErrorId		: UDINT;
END_VAR
VAR
//  INTERNAL VAR
  _AxisREF_P		        		: POINTER TO AXIS_REF;
  _udCalibrationSensor_P  	: POINTER TO UDINT;
  _LineNumber_P             : POINTER TO INT;
  _nAxisTorque_P            : POINTER TO INT;
	_bIsDone                	: BOOL;
  _bIsBusy                	: BOOL;
  _lrActPos                 : LREAL;

//  Request var	BOOL
	bRequestStop		  				: BOOL := FALSE;
	bRequestPowerOn						: BOOL := FALSE;
	bRequestPowerOff					: BOOL := FALSE;
	bRequestHoming						: BOOL := FALSE;
	bRequestReset		  				: BOOL := FALSE;
	bRequestMoveAbso					: BOOL := FALSE;
	bInit               			: BOOL;
	
// FBs
	fbPower				      : MC_Power;
	fbStop				      : MC_Stop;
	fbReset				      : MC_Reset; 
	fbHome				      : MC_Home;
  fbHomeInv				    : MC_Home;
	fbMoveAbso				  : MC_MoveAbsolute;
  fbReadStatus        : MC_ReadStatus;
  fbMoveJog           : MC_Jog;
  fbTimeRetryHomming  : TON := (PT := T#1S);
  fbTimeAbortHoming   : ton := (PT := T#20S);
  fbTimeOutReset  : ton := (PT := T#2S);
  fbTrigErrorMotor    : R_Trig;
  
//Other var
	nStep			          : INT;
  nHistoryStep_AR     : ARRAY[0..C.uiHistoryStep_C] OF INT;
  nLastStep           : INT := -1;
  i                   : INT;
  stHomingOption	    : ST_HomingOptions;
  stHomingInvOption	  : ST_HomingOptions;
  stJogControl        : ST_HmiControlMotor;
  lrSetHomingCheckPos : LREAL;
	lrnOffsetExtractorHoming : LREAL;
	
//  Defect Objet
  objMotorError           : CL_Defect;
  objMoveAbsError         : CL_Defect;
  objMotorResetError      : CL_Defect;
  objMotorPowerError      : CL_Defect;
  objHommingError         : CL_Defect;
  
